REGION Network 42: MB3 Code 4082 - REGOLAZ. BORDATRICE - PASSAGGIO 02 - LATO-OP
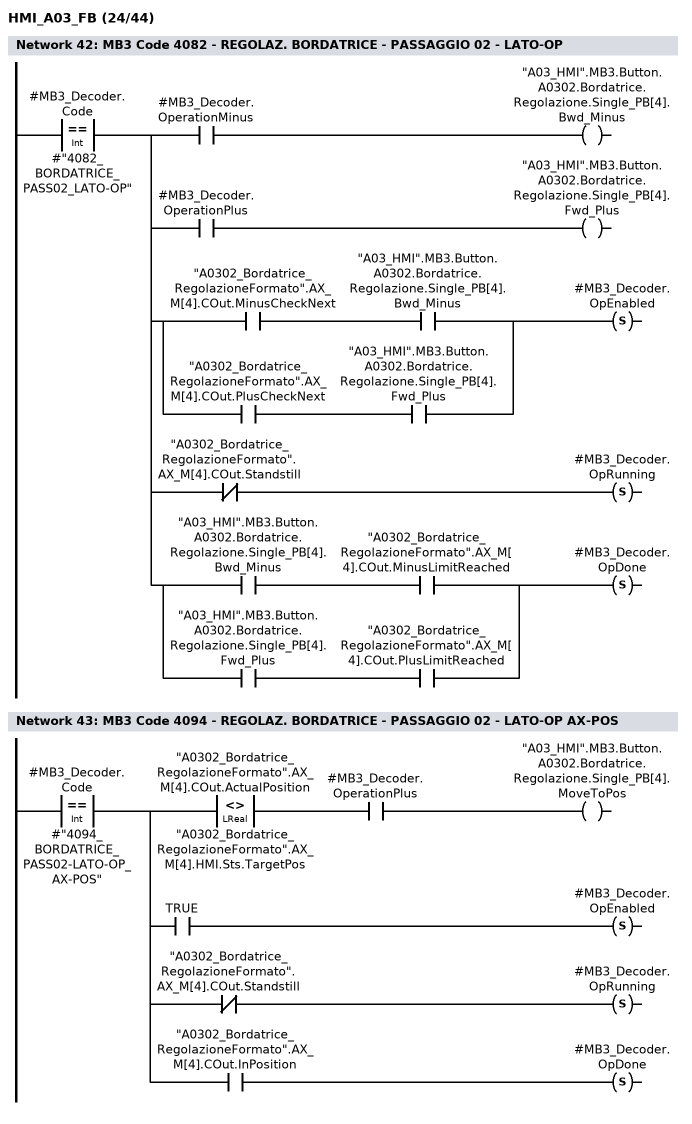
   RUNG wire#powerrail
      { S7_Templates := "SrcType := Int" } EQ_Contact(in1 := #MB3_Decoder.Code, in2 := #"4082_BORDATRICE_PASS02_LATO-OP")
      wire#w1
      Contact( #MB3_Decoder.OperationMinus )
      Coil( "A03_HMI".MB3.Button.A0302.Bordatrice.Regolazione.Single_PB[4].Bwd_Minus )
   END_RUNG
   RUNG wire#w1
      Contact( #MB3_Decoder.OperationPlus )
      Coil( "A03_HMI".MB3.Button.A0302.Bordatrice.Regolazione.Single_PB[4].Fwd_Plus )
   END_RUNG
   RUNG wire#w1
      Contact( "A0302_Bordatrice_RegolazioneFormato".AX_M[4].COut.MinusCheckNext )
      Contact( "A03_HMI".MB3.Button.A0302.Bordatrice.Regolazione.Single_PB[4].Bwd_Minus )
      wire#w2
      S_Coil( #MB3_Decoder.OpEnabled )
   END_RUNG
   RUNG wire#w1
      Contact( "A0302_Bordatrice_RegolazioneFormato".AX_M[4].COut.PlusCheckNext )
      Contact( "A03_HMI".MB3.Button.A0302.Bordatrice.Regolazione.Single_PB[4].Fwd_Plus )
   END_RUNG wire#w2
   RUNG wire#w1
      I_Contact( "A0302_Bordatrice_RegolazioneFormato".AX_M[4].COut.Standstill )
      S_Coil( #MB3_Decoder.OpRunning )
   END_RUNG
   RUNG wire#w1
      Contact( "A03_HMI".MB3.Button.A0302.Bordatrice.Regolazione.Single_PB[4].Bwd_Minus )
      Contact( "A0302_Bordatrice_RegolazioneFormato".AX_M[4].COut.MinusLimitReached )
      wire#w3
      S_Coil( #MB3_Decoder.OpDone )
   END_RUNG
   RUNG wire#w1
      Contact( "A03_HMI".MB3.Button.A0302.Bordatrice.Regolazione.Single_PB[4].Fwd_Plus )
      Contact( "A0302_Bordatrice_RegolazioneFormato".AX_M[4].COut.PlusLimitReached )
   END_RUNG wire#w3
   // the same network as SCL:
   #_w1 := #MB3_Decoder.Code = #"4082_BORDATRICE_PASS02_LATO-OP";
   "A03_HMI".MB3.Button.A0302.Bordatrice.Regolazione.Single_PB[4].Bwd_Minus := #_w1 AND #MB3_Decoder.OperationMinus;
   "A03_HMI".MB3.Button.A0302.Bordatrice.Regolazione.Single_PB[4].Fwd_Plus := #_w1 AND #MB3_Decoder.OperationPlus;
   IF #_w1 AND (("A0302_Bordatrice_RegolazioneFormato".AX_M[4].COut.MinusCheckNext AND "A03_HMI".MB3.Button.A0302.Bordatrice.Regolazione.Single_PB[4].Bwd_Minus) OR ("A0302_Bordatrice_RegolazioneFormato".AX_M[4].COut.PlusCheckNext AND "A03_HMI".MB3.Button.A0302.Bordatrice.Regolazione.Single_PB[4].Fwd_Plus)) THEN
       #MB3_Decoder.OpEnabled := TRUE;
   END_IF;
   IF #_w1 AND NOT "A0302_Bordatrice_RegolazioneFormato".AX_M[4].COut.Standstill THEN
       #MB3_Decoder.OpRunning := TRUE;
   END_IF;
   IF #_w1 AND (("A03_HMI".MB3.Button.A0302.Bordatrice.Regolazione.Single_PB[4].Bwd_Minus AND "A0302_Bordatrice_RegolazioneFormato".AX_M[4].COut.MinusLimitReached) OR ("A03_HMI".MB3.Button.A0302.Bordatrice.Regolazione.Single_PB[4].Fwd_Plus AND "A0302_Bordatrice_RegolazioneFormato".AX_M[4].COut.PlusLimitReached)) THEN
       #MB3_Decoder.OpDone := TRUE;
   END_IF;
END_REGION

REGION Network 43: MB3 Code 4094 - REGOLAZ. BORDATRICE - PASSAGGIO 02 - LATO-OP AX-POS
   RUNG wire#powerrail
      { S7_Templates := "SrcType := Int" } EQ_Contact(in1 := #MB3_Decoder.Code, in2 := #"4094_BORDATRICE_PASS02-LATO-OP_AX-POS")
      wire#w1
      { S7_Templates := "SrcType := LReal" } NE_Contact(in1 := "A0302_Bordatrice_RegolazioneFormato".AX_M[4].COut.ActualPosition, in2 := "A0302_Bordatrice_RegolazioneFormato".AX_M[4].HMI.Sts.TargetPos)
      Contact( #MB3_Decoder.OperationPlus )
      Coil( "A03_HMI".MB3.Button.A0302.Bordatrice.Regolazione.Single_PB[4].MoveToPos )
   END_RUNG
   RUNG wire#w1
      Contact( TRUE )
      S_Coil( #MB3_Decoder.OpEnabled )
   END_RUNG
   RUNG wire#w1
      I_Contact( "A0302_Bordatrice_RegolazioneFormato".AX_M[4].COut.Standstill )
      S_Coil( #MB3_Decoder.OpRunning )
   END_RUNG
   RUNG wire#w1
      Contact( "A0302_Bordatrice_RegolazioneFormato".AX_M[4].COut.InPosition )
      S_Coil( #MB3_Decoder.OpDone )
   END_RUNG
   // the same network as SCL:
   #_w1 := #MB3_Decoder.Code = #"4094_BORDATRICE_PASS02-LATO-OP_AX-POS";
   "A03_HMI".MB3.Button.A0302.Bordatrice.Regolazione.Single_PB[4].MoveToPos := #_w1 AND ("A0302_Bordatrice_RegolazioneFormato".AX_M[4].COut.ActualPosition <> "A0302_Bordatrice_RegolazioneFormato".AX_M[4].HMI.Sts.TargetPos) AND #MB3_Decoder.OperationPlus;
   IF #_w1 AND TRUE THEN #MB3_Decoder.OpEnabled := TRUE; END_IF;
   IF #_w1 AND NOT "A0302_Bordatrice_RegolazioneFormato".AX_M[4].COut.Standstill THEN
       #MB3_Decoder.OpRunning := TRUE;
   END_IF;
   IF #_w1 AND "A0302_Bordatrice_RegolazioneFormato".AX_M[4].COut.InPosition THEN
       #MB3_Decoder.OpDone := TRUE;
   END_IF;
END_REGION

REGION Network 44: MB3 Code 4083 - REGOLAZ. BORDATRICE - PASSAGGIO 02 - LATO-MOT
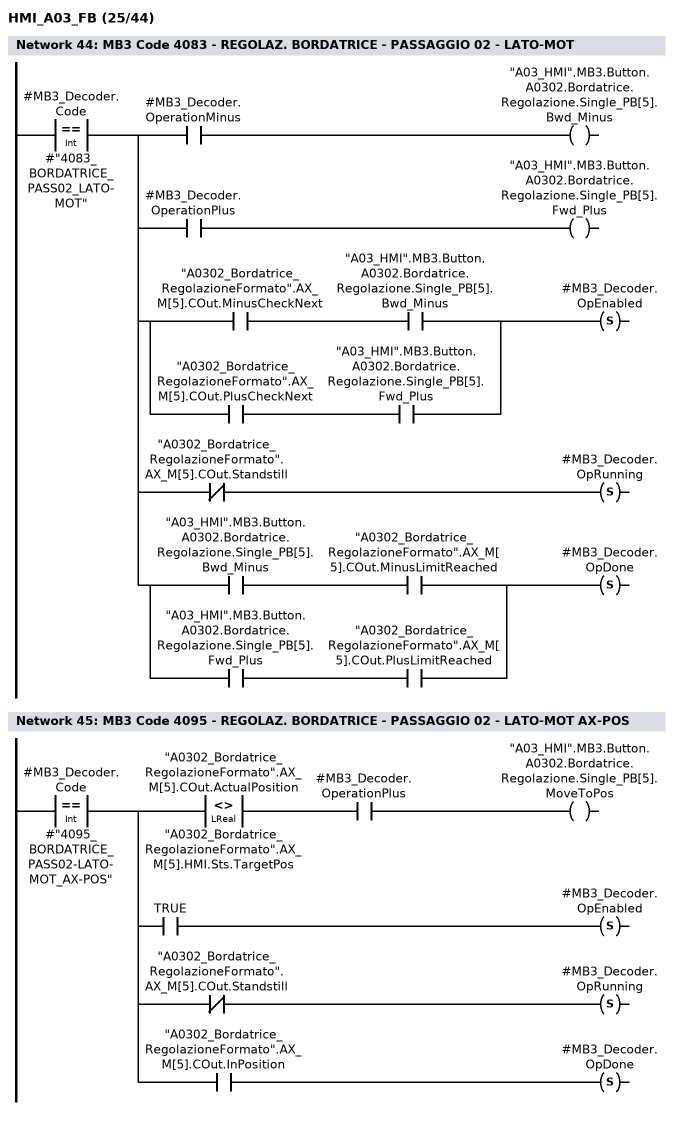
   RUNG wire#powerrail
      { S7_Templates := "SrcType := Int" } EQ_Contact(in1 := #MB3_Decoder.Code, in2 := #"4083_BORDATRICE_PASS02_LATO-MOT")
      wire#w1
      Contact( #MB3_Decoder.OperationMinus )
      Coil( "A03_HMI".MB3.Button.A0302.Bordatrice.Regolazione.Single_PB[5].Bwd_Minus )
   END_RUNG
   RUNG wire#w1
      Contact( #MB3_Decoder.OperationPlus )
      Coil( "A03_HMI".MB3.Button.A0302.Bordatrice.Regolazione.Single_PB[5].Fwd_Plus )
   END_RUNG
   RUNG wire#w1
      Contact( "A0302_Bordatrice_RegolazioneFormato".AX_M[5].COut.MinusCheckNext )
      Contact( "A03_HMI".MB3.Button.A0302.Bordatrice.Regolazione.Single_PB[5].Bwd_Minus )
      wire#w2
      S_Coil( #MB3_Decoder.OpEnabled )
   END_RUNG
   RUNG wire#w1
      Contact( "A0302_Bordatrice_RegolazioneFormato".AX_M[5].COut.PlusCheckNext )
      Contact( "A03_HMI".MB3.Button.A0302.Bordatrice.Regolazione.Single_PB[5].Fwd_Plus )
   END_RUNG wire#w2
   RUNG wire#w1
      I_Contact( "A0302_Bordatrice_RegolazioneFormato".AX_M[5].COut.Standstill )
      S_Coil( #MB3_Decoder.OpRunning )
   END_RUNG
   RUNG wire#w1
      Contact( "A03_HMI".MB3.Button.A0302.Bordatrice.Regolazione.Single_PB[5].Bwd_Minus )
      Contact( "A0302_Bordatrice_RegolazioneFormato".AX_M[5].COut.MinusLimitReached )
      wire#w3
      S_Coil( #MB3_Decoder.OpDone )
   END_RUNG
   RUNG wire#w1
      Contact( "A03_HMI".MB3.Button.A0302.Bordatrice.Regolazione.Single_PB[5].Fwd_Plus )
      Contact( "A0302_Bordatrice_RegolazioneFormato".AX_M[5].COut.PlusLimitReached )
   END_RUNG wire#w3
   // the same network as SCL:
   #_w1 := #MB3_Decoder.Code = #"4083_BORDATRICE_PASS02_LATO-MOT";
   "A03_HMI".MB3.Button.A0302.Bordatrice.Regolazione.Single_PB[5].Bwd_Minus := #_w1 AND #MB3_Decoder.OperationMinus;
   "A03_HMI".MB3.Button.A0302.Bordatrice.Regolazione.Single_PB[5].Fwd_Plus := #_w1 AND #MB3_Decoder.OperationPlus;
   IF #_w1 AND (("A0302_Bordatrice_RegolazioneFormato".AX_M[5].COut.MinusCheckNext AND "A03_HMI".MB3.Button.A0302.Bordatrice.Regolazione.Single_PB[5].Bwd_Minus) OR ("A0302_Bordatrice_RegolazioneFormato".AX_M[5].COut.PlusCheckNext AND "A03_HMI".MB3.Button.A0302.Bordatrice.Regolazione.Single_PB[5].Fwd_Plus)) THEN
       #MB3_Decoder.OpEnabled := TRUE;
   END_IF;
   IF #_w1 AND NOT "A0302_Bordatrice_RegolazioneFormato".AX_M[5].COut.Standstill THEN
       #MB3_Decoder.OpRunning := TRUE;
   END_IF;
   IF #_w1 AND (("A03_HMI".MB3.Button.A0302.Bordatrice.Regolazione.Single_PB[5].Bwd_Minus AND "A0302_Bordatrice_RegolazioneFormato".AX_M[5].COut.MinusLimitReached) OR ("A03_HMI".MB3.Button.A0302.Bordatrice.Regolazione.Single_PB[5].Fwd_Plus AND "A0302_Bordatrice_RegolazioneFormato".AX_M[5].COut.PlusLimitReached)) THEN
       #MB3_Decoder.OpDone := TRUE;
   END_IF;
END_REGION

REGION Network 45: MB3 Code 4095 - REGOLAZ. BORDATRICE - PASSAGGIO 02 - LATO-MOT AX-POS
   RUNG wire#powerrail
      { S7_Templates := "SrcType := Int" } EQ_Contact(in1 := #MB3_Decoder.Code, in2 := #"4095_BORDATRICE_PASS02-LATO-MOT_AX-POS")
      wire#w1
      { S7_Templates := "SrcType := LReal" } NE_Contact(in1 := "A0302_Bordatrice_RegolazioneFormato".AX_M[5].COut.ActualPosition, in2 := "A0302_Bordatrice_RegolazioneFormato".AX_M[5].HMI.Sts.TargetPos)
      Contact( #MB3_Decoder.OperationPlus )
      Coil( "A03_HMI".MB3.Button.A0302.Bordatrice.Regolazione.Single_PB[5].MoveToPos )
   END_RUNG
   RUNG wire#w1
      Contact( TRUE )
      S_Coil( #MB3_Decoder.OpEnabled )
   END_RUNG
   RUNG wire#w1
      I_Contact( "A0302_Bordatrice_RegolazioneFormato".AX_M[5].COut.Standstill )
      S_Coil( #MB3_Decoder.OpRunning )
   END_RUNG
   RUNG wire#w1
      Contact( "A0302_Bordatrice_RegolazioneFormato".AX_M[5].COut.InPosition )
      S_Coil( #MB3_Decoder.OpDone )
   END_RUNG
   // the same network as SCL:
   #_w1 := #MB3_Decoder.Code = #"4095_BORDATRICE_PASS02-LATO-MOT_AX-POS";
   "A03_HMI".MB3.Button.A0302.Bordatrice.Regolazione.Single_PB[5].MoveToPos := #_w1 AND ("A0302_Bordatrice_RegolazioneFormato".AX_M[5].COut.ActualPosition <> "A0302_Bordatrice_RegolazioneFormato".AX_M[5].HMI.Sts.TargetPos) AND #MB3_Decoder.OperationPlus;
   IF #_w1 AND TRUE THEN #MB3_Decoder.OpEnabled := TRUE; END_IF;
   IF #_w1 AND NOT "A0302_Bordatrice_RegolazioneFormato".AX_M[5].COut.Standstill THEN
       #MB3_Decoder.OpRunning := TRUE;
   END_IF;
   IF #_w1 AND "A0302_Bordatrice_RegolazioneFormato".AX_M[5].COut.InPosition THEN
       #MB3_Decoder.OpDone := TRUE;
   END_IF;
END_REGION

REGION Network 46: MB3 Code 4036 - REGOLAZ. BORDATRICE - PASSAGGIO 03 - COMBO
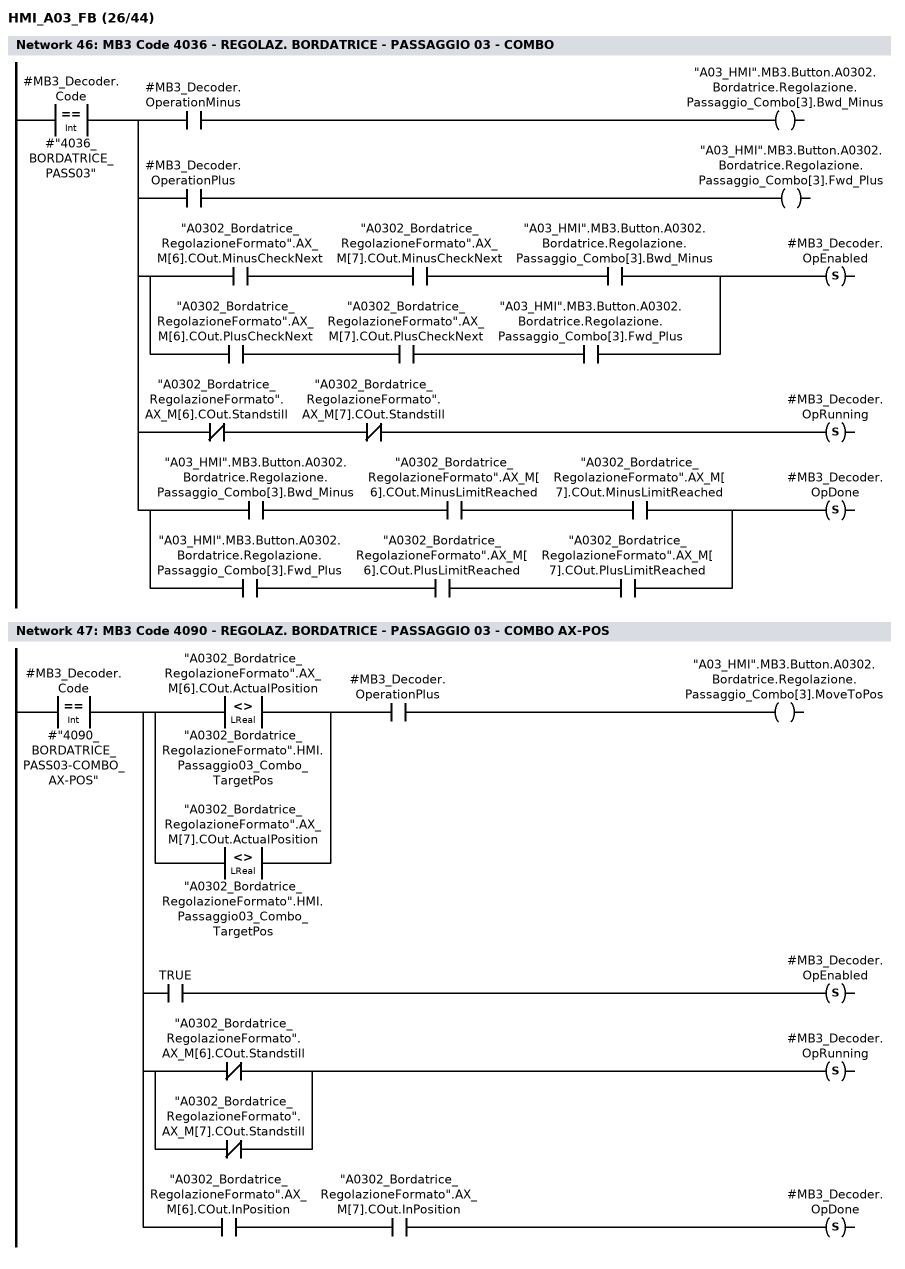
   RUNG wire#powerrail
      { S7_Templates := "SrcType := Int" } EQ_Contact(in1 := #MB3_Decoder.Code, in2 := #"4036_BORDATRICE_PASS03")
      wire#w1
      Contact( #MB3_Decoder.OperationMinus )
      Coil( "A03_HMI".MB3.Button.A0302.Bordatrice.Regolazione.Passaggio_Combo[3].Bwd_Minus )
   END_RUNG
   RUNG wire#w1
      Contact( #MB3_Decoder.OperationPlus )
      Coil( "A03_HMI".MB3.Button.A0302.Bordatrice.Regolazione.Passaggio_Combo[3].Fwd_Plus )
   END_RUNG
   RUNG wire#w1
      Contact( "A0302_Bordatrice_RegolazioneFormato".AX_M[6].COut.MinusCheckNext )
      Contact( "A0302_Bordatrice_RegolazioneFormato".AX_M[7].COut.MinusCheckNext )
      Contact( "A03_HMI".MB3.Button.A0302.Bordatrice.Regolazione.Passaggio_Combo[3].Bwd_Minus )
      wire#w2
      S_Coil( #MB3_Decoder.OpEnabled )
   END_RUNG
   RUNG wire#w1
      Contact( "A0302_Bordatrice_RegolazioneFormato".AX_M[6].COut.PlusCheckNext )
      Contact( "A0302_Bordatrice_RegolazioneFormato".AX_M[7].COut.PlusCheckNext )
      Contact( "A03_HMI".MB3.Button.A0302.Bordatrice.Regolazione.Passaggio_Combo[3].Fwd_Plus )
   END_RUNG wire#w2
   RUNG wire#w1
      I_Contact( "A0302_Bordatrice_RegolazioneFormato".AX_M[6].COut.Standstill )
      I_Contact( "A0302_Bordatrice_RegolazioneFormato".AX_M[7].COut.Standstill )
      S_Coil( #MB3_Decoder.OpRunning )
   END_RUNG
   RUNG wire#w1
      Contact( "A03_HMI".MB3.Button.A0302.Bordatrice.Regolazione.Passaggio_Combo[3].Bwd_Minus )
      Contact( "A0302_Bordatrice_RegolazioneFormato".AX_M[6].COut.MinusLimitReached )
      Contact( "A0302_Bordatrice_RegolazioneFormato".AX_M[7].COut.MinusLimitReached )
      wire#w3
      S_Coil( #MB3_Decoder.OpDone )
   END_RUNG
   RUNG wire#w1
      Contact( "A03_HMI".MB3.Button.A0302.Bordatrice.Regolazione.Passaggio_Combo[3].Fwd_Plus )
      Contact( "A0302_Bordatrice_RegolazioneFormato".AX_M[6].COut.PlusLimitReached )
      Contact( "A0302_Bordatrice_RegolazioneFormato".AX_M[7].COut.PlusLimitReached )
   END_RUNG wire#w3
   // the same network as SCL:
   #_w1 := #MB3_Decoder.Code = #"4036_BORDATRICE_PASS03";
   "A03_HMI".MB3.Button.A0302.Bordatrice.Regolazione.Passaggio_Combo[3].Bwd_Minus := #_w1 AND #MB3_Decoder.OperationMinus;
   "A03_HMI".MB3.Button.A0302.Bordatrice.Regolazione.Passaggio_Combo[3].Fwd_Plus := #_w1 AND #MB3_Decoder.OperationPlus;
   IF #_w1 AND (("A0302_Bordatrice_RegolazioneFormato".AX_M[6].COut.MinusCheckNext AND "A0302_Bordatrice_RegolazioneFormato".AX_M[7].COut.MinusCheckNext AND "A03_HMI".MB3.Button.A0302.Bordatrice.Regolazione.Passaggio_Combo[3].Bwd_Minus) OR ("A0302_Bordatrice_RegolazioneFormato".AX_M[6].COut.PlusCheckNext AND "A0302_Bordatrice_RegolazioneFormato".AX_M[7].COut.PlusCheckNext AND "A03_HMI".MB3.Button.A0302.Bordatrice.Regolazione.Passaggio_Combo[3].Fwd_Plus)) THEN
       #MB3_Decoder.OpEnabled := TRUE;
   END_IF;
   IF #_w1 AND NOT "A0302_Bordatrice_RegolazioneFormato".AX_M[6].COut.Standstill AND NOT "A0302_Bordatrice_RegolazioneFormato".AX_M[7].COut.Standstill THEN
       #MB3_Decoder.OpRunning := TRUE;
   END_IF;
   IF #_w1 AND (("A03_HMI".MB3.Button.A0302.Bordatrice.Regolazione.Passaggio_Combo[3].Bwd_Minus AND "A0302_Bordatrice_RegolazioneFormato".AX_M[6].COut.MinusLimitReached AND "A0302_Bordatrice_RegolazioneFormato".AX_M[7].COut.MinusLimitReached) OR ("A03_HMI".MB3.Button.A0302.Bordatrice.Regolazione.Passaggio_Combo[3].Fwd_Plus AND "A0302_Bordatrice_RegolazioneFormato".AX_M[6].COut.PlusLimitReached AND "A0302_Bordatrice_RegolazioneFormato".AX_M[7].COut.PlusLimitReached)) THEN
       #MB3_Decoder.OpDone := TRUE;
   END_IF;
END_REGION

REGION Network 47: MB3 Code 4090 - REGOLAZ. BORDATRICE - PASSAGGIO 03 - COMBO AX-POS
   RUNG wire#powerrail
      { S7_Templates := "SrcType := Int" } EQ_Contact(in1 := #MB3_Decoder.Code, in2 := #"4090_BORDATRICE_PASS03-COMBO_AX-POS")
      wire#w1
      { S7_Templates := "SrcType := LReal" } NE_Contact(in1 := "A0302_Bordatrice_RegolazioneFormato".AX_M[6].COut.ActualPosition, in2 := "A0302_Bordatrice_RegolazioneFormato".HMI.Passaggio03_Combo_TargetPos)
      wire#w2
      Contact( #MB3_Decoder.OperationPlus )
      Coil( "A03_HMI".MB3.Button.A0302.Bordatrice.Regolazione.Passaggio_Combo[3].MoveToPos )
   END_RUNG
   RUNG wire#w1
      { S7_Templates := "SrcType := LReal" } NE_Contact(in1 := "A0302_Bordatrice_RegolazioneFormato".AX_M[7].COut.ActualPosition, in2 := "A0302_Bordatrice_RegolazioneFormato".HMI.Passaggio03_Combo_TargetPos)
   END_RUNG wire#w2
   RUNG wire#w1
      Contact( TRUE )
      S_Coil( #MB3_Decoder.OpEnabled )
   END_RUNG
   RUNG wire#w1
      I_Contact( "A0302_Bordatrice_RegolazioneFormato".AX_M[6].COut.Standstill )
      wire#w3
      S_Coil( #MB3_Decoder.OpRunning )
   END_RUNG
   RUNG wire#w1
      I_Contact( "A0302_Bordatrice_RegolazioneFormato".AX_M[7].COut.Standstill )
   END_RUNG wire#w3
   RUNG wire#w1
      Contact( "A0302_Bordatrice_RegolazioneFormato".AX_M[6].COut.InPosition )
      Contact( "A0302_Bordatrice_RegolazioneFormato".AX_M[7].COut.InPosition )
      S_Coil( #MB3_Decoder.OpDone )
   END_RUNG
   // the same network as SCL:
   #_w1 := #MB3_Decoder.Code = #"4090_BORDATRICE_PASS03-COMBO_AX-POS";
   "A03_HMI".MB3.Button.A0302.Bordatrice.Regolazione.Passaggio_Combo[3].MoveToPos := #_w1 AND (("A0302_Bordatrice_RegolazioneFormato".AX_M[6].COut.ActualPosition <> "A0302_Bordatrice_RegolazioneFormato".HMI.Passaggio03_Combo_TargetPos) OR ("A0302_Bordatrice_RegolazioneFormato".AX_M[7].COut.ActualPosition <> "A0302_Bordatrice_RegolazioneFormato".HMI.Passaggio03_Combo_TargetPos)) AND #MB3_Decoder.OperationPlus;
   IF #_w1 AND TRUE THEN #MB3_Decoder.OpEnabled := TRUE; END_IF;
   IF #_w1 AND (NOT "A0302_Bordatrice_RegolazioneFormato".AX_M[6].COut.Standstill OR NOT "A0302_Bordatrice_RegolazioneFormato".AX_M[7].COut.Standstill) THEN
       #MB3_Decoder.OpRunning := TRUE;
   END_IF;
   IF #_w1 AND "A0302_Bordatrice_RegolazioneFormato".AX_M[6].COut.InPosition AND "A0302_Bordatrice_RegolazioneFormato".AX_M[7].COut.InPosition THEN
       #MB3_Decoder.OpDone := TRUE;
   END_IF;
END_REGION

REGION Network 48: MB3 Code 4084 - REGOLAZ. BORDATRICE - PASSAGGIO 03 - LATO-OP
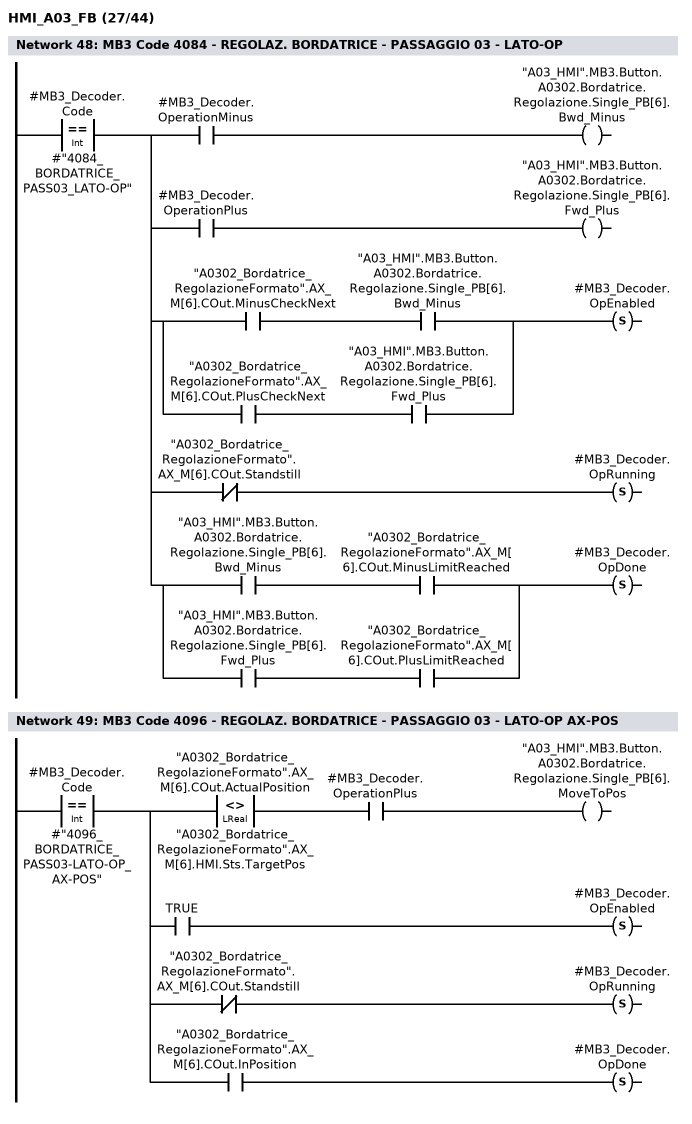
   RUNG wire#powerrail
      { S7_Templates := "SrcType := Int" } EQ_Contact(in1 := #MB3_Decoder.Code, in2 := #"4084_BORDATRICE_PASS03_LATO-OP")
      wire#w1
      Contact( #MB3_Decoder.OperationMinus )
      Coil( "A03_HMI".MB3.Button.A0302.Bordatrice.Regolazione.Single_PB[6].Bwd_Minus )
   END_RUNG
   RUNG wire#w1
      Contact( #MB3_Decoder.OperationPlus )
      Coil( "A03_HMI".MB3.Button.A0302.Bordatrice.Regolazione.Single_PB[6].Fwd_Plus )
   END_RUNG
   RUNG wire#w1
      Contact( "A0302_Bordatrice_RegolazioneFormato".AX_M[6].COut.MinusCheckNext )
      Contact( "A03_HMI".MB3.Button.A0302.Bordatrice.Regolazione.Single_PB[6].Bwd_Minus )
      wire#w2
      S_Coil( #MB3_Decoder.OpEnabled )
   END_RUNG
   RUNG wire#w1
      Contact( "A0302_Bordatrice_RegolazioneFormato".AX_M[6].COut.PlusCheckNext )
      Contact( "A03_HMI".MB3.Button.A0302.Bordatrice.Regolazione.Single_PB[6].Fwd_Plus )
   END_RUNG wire#w2
   RUNG wire#w1
      I_Contact( "A0302_Bordatrice_RegolazioneFormato".AX_M[6].COut.Standstill )
      S_Coil( #MB3_Decoder.OpRunning )
   END_RUNG
   RUNG wire#w1
      Contact( "A03_HMI".MB3.Button.A0302.Bordatrice.Regolazione.Single_PB[6].Bwd_Minus )
      Contact( "A0302_Bordatrice_RegolazioneFormato".AX_M[6].COut.MinusLimitReached )
      wire#w3
      S_Coil( #MB3_Decoder.OpDone )
   END_RUNG
   RUNG wire#w1
      Contact( "A03_HMI".MB3.Button.A0302.Bordatrice.Regolazione.Single_PB[6].Fwd_Plus )
      Contact( "A0302_Bordatrice_RegolazioneFormato".AX_M[6].COut.PlusLimitReached )
   END_RUNG wire#w3
   // the same network as SCL:
   #_w1 := #MB3_Decoder.Code = #"4084_BORDATRICE_PASS03_LATO-OP";
   "A03_HMI".MB3.Button.A0302.Bordatrice.Regolazione.Single_PB[6].Bwd_Minus := #_w1 AND #MB3_Decoder.OperationMinus;
   "A03_HMI".MB3.Button.A0302.Bordatrice.Regolazione.Single_PB[6].Fwd_Plus := #_w1 AND #MB3_Decoder.OperationPlus;
   IF #_w1 AND (("A0302_Bordatrice_RegolazioneFormato".AX_M[6].COut.MinusCheckNext AND "A03_HMI".MB3.Button.A0302.Bordatrice.Regolazione.Single_PB[6].Bwd_Minus) OR ("A0302_Bordatrice_RegolazioneFormato".AX_M[6].COut.PlusCheckNext AND "A03_HMI".MB3.Button.A0302.Bordatrice.Regolazione.Single_PB[6].Fwd_Plus)) THEN
       #MB3_Decoder.OpEnabled := TRUE;
   END_IF;
   IF #_w1 AND NOT "A0302_Bordatrice_RegolazioneFormato".AX_M[6].COut.Standstill THEN
       #MB3_Decoder.OpRunning := TRUE;
   END_IF;
   IF #_w1 AND (("A03_HMI".MB3.Button.A0302.Bordatrice.Regolazione.Single_PB[6].Bwd_Minus AND "A0302_Bordatrice_RegolazioneFormato".AX_M[6].COut.MinusLimitReached) OR ("A03_HMI".MB3.Button.A0302.Bordatrice.Regolazione.Single_PB[6].Fwd_Plus AND "A0302_Bordatrice_RegolazioneFormato".AX_M[6].COut.PlusLimitReached)) THEN
       #MB3_Decoder.OpDone := TRUE;
   END_IF;
END_REGION

REGION Network 49: MB3 Code 4096 - REGOLAZ. BORDATRICE - PASSAGGIO 03 - LATO-OP AX-POS
   RUNG wire#powerrail
      { S7_Templates := "SrcType := Int" } EQ_Contact(in1 := #MB3_Decoder.Code, in2 := #"4096_BORDATRICE_PASS03-LATO-OP_AX-POS")
      wire#w1
      { S7_Templates := "SrcType := LReal" } NE_Contact(in1 := "A0302_Bordatrice_RegolazioneFormato".AX_M[6].COut.ActualPosition, in2 := "A0302_Bordatrice_RegolazioneFormato".AX_M[6].HMI.Sts.TargetPos)
      Contact( #MB3_Decoder.OperationPlus )
      Coil( "A03_HMI".MB3.Button.A0302.Bordatrice.Regolazione.Single_PB[6].MoveToPos )
   END_RUNG
   RUNG wire#w1
      Contact( TRUE )
      S_Coil( #MB3_Decoder.OpEnabled )
   END_RUNG
   RUNG wire#w1
      I_Contact( "A0302_Bordatrice_RegolazioneFormato".AX_M[6].COut.Standstill )
      S_Coil( #MB3_Decoder.OpRunning )
   END_RUNG
   RUNG wire#w1
      Contact( "A0302_Bordatrice_RegolazioneFormato".AX_M[6].COut.InPosition )
      S_Coil( #MB3_Decoder.OpDone )
   END_RUNG
   // the same network as SCL:
   #_w1 := #MB3_Decoder.Code = #"4096_BORDATRICE_PASS03-LATO-OP_AX-POS";
   "A03_HMI".MB3.Button.A0302.Bordatrice.Regolazione.Single_PB[6].MoveToPos := #_w1 AND ("A0302_Bordatrice_RegolazioneFormato".AX_M[6].COut.ActualPosition <> "A0302_Bordatrice_RegolazioneFormato".AX_M[6].HMI.Sts.TargetPos) AND #MB3_Decoder.OperationPlus;
   IF #_w1 AND TRUE THEN #MB3_Decoder.OpEnabled := TRUE; END_IF;
   IF #_w1 AND NOT "A0302_Bordatrice_RegolazioneFormato".AX_M[6].COut.Standstill THEN
       #MB3_Decoder.OpRunning := TRUE;
   END_IF;
   IF #_w1 AND "A0302_Bordatrice_RegolazioneFormato".AX_M[6].COut.InPosition THEN
       #MB3_Decoder.OpDone := TRUE;
   END_IF;
END_REGION

REGION Network 50: MB3 Code 4085 - REGOLAZ. BORDATRICE - PASSAGGIO 03 - LATO-MOT
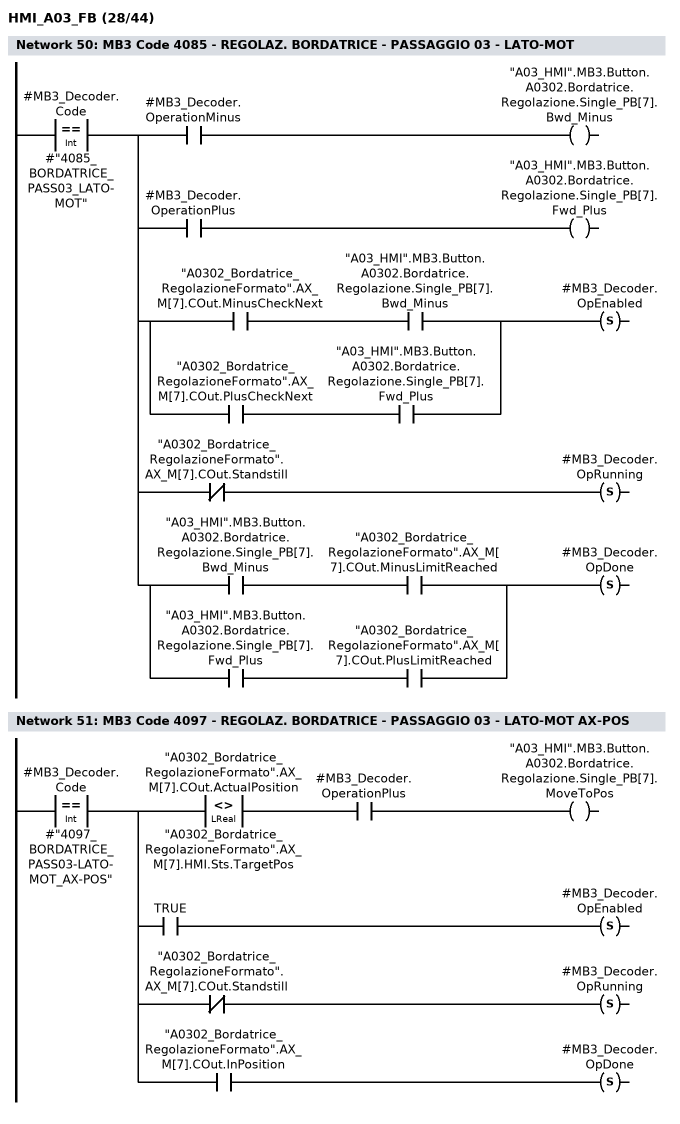
   RUNG wire#powerrail
      { S7_Templates := "SrcType := Int" } EQ_Contact(in1 := #MB3_Decoder.Code, in2 := #"4085_BORDATRICE_PASS03_LATO-MOT")
      wire#w1
      Contact( #MB3_Decoder.OperationMinus )
      Coil( "A03_HMI".MB3.Button.A0302.Bordatrice.Regolazione.Single_PB[7].Bwd_Minus )
   END_RUNG
   RUNG wire#w1
      Contact( #MB3_Decoder.OperationPlus )
      Coil( "A03_HMI".MB3.Button.A0302.Bordatrice.Regolazione.Single_PB[7].Fwd_Plus )
   END_RUNG
   RUNG wire#w1
      Contact( "A0302_Bordatrice_RegolazioneFormato".AX_M[7].COut.MinusCheckNext )
      Contact( "A03_HMI".MB3.Button.A0302.Bordatrice.Regolazione.Single_PB[7].Bwd_Minus )
      wire#w2
      S_Coil( #MB3_Decoder.OpEnabled )
   END_RUNG
   RUNG wire#w1
      Contact( "A0302_Bordatrice_RegolazioneFormato".AX_M[7].COut.PlusCheckNext )
      Contact( "A03_HMI".MB3.Button.A0302.Bordatrice.Regolazione.Single_PB[7].Fwd_Plus )
   END_RUNG wire#w2
   RUNG wire#w1
      I_Contact( "A0302_Bordatrice_RegolazioneFormato".AX_M[7].COut.Standstill )
      S_Coil( #MB3_Decoder.OpRunning )
   END_RUNG
   RUNG wire#w1
      Contact( "A03_HMI".MB3.Button.A0302.Bordatrice.Regolazione.Single_PB[7].Bwd_Minus )
      Contact( "A0302_Bordatrice_RegolazioneFormato".AX_M[7].COut.MinusLimitReached )
      wire#w3
      S_Coil( #MB3_Decoder.OpDone )
   END_RUNG
   RUNG wire#w1
      Contact( "A03_HMI".MB3.Button.A0302.Bordatrice.Regolazione.Single_PB[7].Fwd_Plus )
      Contact( "A0302_Bordatrice_RegolazioneFormato".AX_M[7].COut.PlusLimitReached )
   END_RUNG wire#w3
   // the same network as SCL:
   #_w1 := #MB3_Decoder.Code = #"4085_BORDATRICE_PASS03_LATO-MOT";
   "A03_HMI".MB3.Button.A0302.Bordatrice.Regolazione.Single_PB[7].Bwd_Minus := #_w1 AND #MB3_Decoder.OperationMinus;
   "A03_HMI".MB3.Button.A0302.Bordatrice.Regolazione.Single_PB[7].Fwd_Plus := #_w1 AND #MB3_Decoder.OperationPlus;
   IF #_w1 AND (("A0302_Bordatrice_RegolazioneFormato".AX_M[7].COut.MinusCheckNext AND "A03_HMI".MB3.Button.A0302.Bordatrice.Regolazione.Single_PB[7].Bwd_Minus) OR ("A0302_Bordatrice_RegolazioneFormato".AX_M[7].COut.PlusCheckNext AND "A03_HMI".MB3.Button.A0302.Bordatrice.Regolazione.Single_PB[7].Fwd_Plus)) THEN
       #MB3_Decoder.OpEnabled := TRUE;
   END_IF;
   IF #_w1 AND NOT "A0302_Bordatrice_RegolazioneFormato".AX_M[7].COut.Standstill THEN
       #MB3_Decoder.OpRunning := TRUE;
   END_IF;
   IF #_w1 AND (("A03_HMI".MB3.Button.A0302.Bordatrice.Regolazione.Single_PB[7].Bwd_Minus AND "A0302_Bordatrice_RegolazioneFormato".AX_M[7].COut.MinusLimitReached) OR ("A03_HMI".MB3.Button.A0302.Bordatrice.Regolazione.Single_PB[7].Fwd_Plus AND "A0302_Bordatrice_RegolazioneFormato".AX_M[7].COut.PlusLimitReached)) THEN
       #MB3_Decoder.OpDone := TRUE;
   END_IF;
END_REGION

REGION Network 51: MB3 Code 4097 - REGOLAZ. BORDATRICE - PASSAGGIO 03 - LATO-MOT AX-POS
   RUNG wire#powerrail
      { S7_Templates := "SrcType := Int" } EQ_Contact(in1 := #MB3_Decoder.Code, in2 := #"4097_BORDATRICE_PASS03-LATO-MOT_AX-POS")
      wire#w1
      { S7_Templates := "SrcType := LReal" } NE_Contact(in1 := "A0302_Bordatrice_RegolazioneFormato".AX_M[7].COut.ActualPosition, in2 := "A0302_Bordatrice_RegolazioneFormato".AX_M[7].HMI.Sts.TargetPos)
      Contact( #MB3_Decoder.OperationPlus )
      Coil( "A03_HMI".MB3.Button.A0302.Bordatrice.Regolazione.Single_PB[7].MoveToPos )
   END_RUNG
   RUNG wire#w1
      Contact( TRUE )
      S_Coil( #MB3_Decoder.OpEnabled )
   END_RUNG
   RUNG wire#w1
      I_Contact( "A0302_Bordatrice_RegolazioneFormato".AX_M[7].COut.Standstill )
      S_Coil( #MB3_Decoder.OpRunning )
   END_RUNG
   RUNG wire#w1
      Contact( "A0302_Bordatrice_RegolazioneFormato".AX_M[7].COut.InPosition )
      S_Coil( #MB3_Decoder.OpDone )
   END_RUNG
   // the same network as SCL:
   #_w1 := #MB3_Decoder.Code = #"4097_BORDATRICE_PASS03-LATO-MOT_AX-POS";
   "A03_HMI".MB3.Button.A0302.Bordatrice.Regolazione.Single_PB[7].MoveToPos := #_w1 AND ("A0302_Bordatrice_RegolazioneFormato".AX_M[7].COut.ActualPosition <> "A0302_Bordatrice_RegolazioneFormato".AX_M[7].HMI.Sts.TargetPos) AND #MB3_Decoder.OperationPlus;
   IF #_w1 AND TRUE THEN #MB3_Decoder.OpEnabled := TRUE; END_IF;
   IF #_w1 AND NOT "A0302_Bordatrice_RegolazioneFormato".AX_M[7].COut.Standstill THEN
       #MB3_Decoder.OpRunning := TRUE;
   END_IF;
   IF #_w1 AND "A0302_Bordatrice_RegolazioneFormato".AX_M[7].COut.InPosition THEN
       #MB3_Decoder.OpDone := TRUE;
   END_IF;
END_REGION

REGION Network 52: MB3 Code 4037 - REGOLAZ. BORDATRICE - PASSAGGIO 04 - COMBO
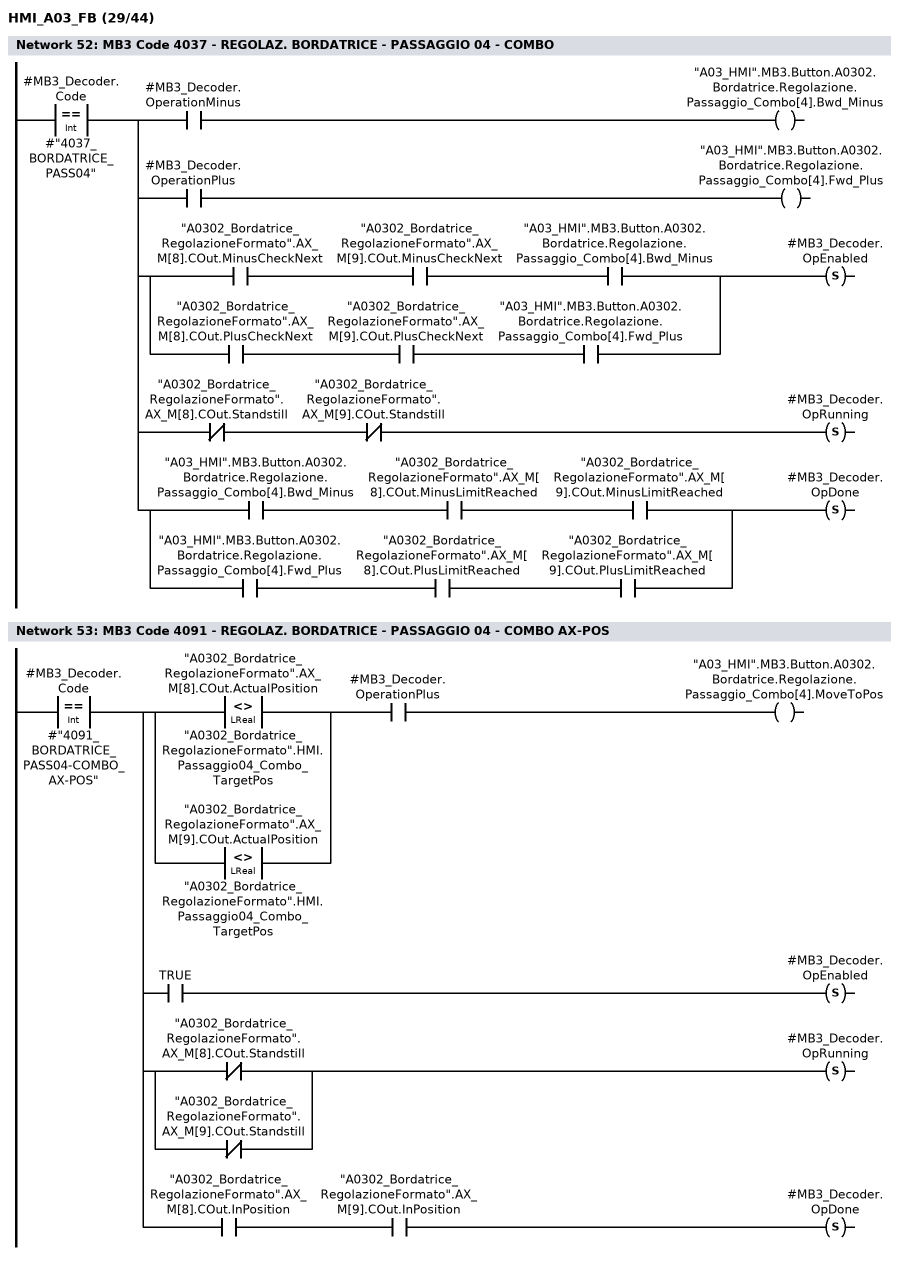
   RUNG wire#powerrail
      { S7_Templates := "SrcType := Int" } EQ_Contact(in1 := #MB3_Decoder.Code, in2 := #"4037_BORDATRICE_PASS04")
      wire#w1
      Contact( #MB3_Decoder.OperationMinus )
      Coil( "A03_HMI".MB3.Button.A0302.Bordatrice.Regolazione.Passaggio_Combo[4].Bwd_Minus )
   END_RUNG
   RUNG wire#w1
      Contact( #MB3_Decoder.OperationPlus )
      Coil( "A03_HMI".MB3.Button.A0302.Bordatrice.Regolazione.Passaggio_Combo[4].Fwd_Plus )
   END_RUNG
   RUNG wire#w1
      Contact( "A0302_Bordatrice_RegolazioneFormato".AX_M[8].COut.MinusCheckNext )
      Contact( "A0302_Bordatrice_RegolazioneFormato".AX_M[9].COut.MinusCheckNext )
      Contact( "A03_HMI".MB3.Button.A0302.Bordatrice.Regolazione.Passaggio_Combo[4].Bwd_Minus )
      wire#w2
      S_Coil( #MB3_Decoder.OpEnabled )
   END_RUNG
   RUNG wire#w1
      Contact( "A0302_Bordatrice_RegolazioneFormato".AX_M[8].COut.PlusCheckNext )
      Contact( "A0302_Bordatrice_RegolazioneFormato".AX_M[9].COut.PlusCheckNext )
      Contact( "A03_HMI".MB3.Button.A0302.Bordatrice.Regolazione.Passaggio_Combo[4].Fwd_Plus )
   END_RUNG wire#w2
   RUNG wire#w1
      I_Contact( "A0302_Bordatrice_RegolazioneFormato".AX_M[8].COut.Standstill )
      I_Contact( "A0302_Bordatrice_RegolazioneFormato".AX_M[9].COut.Standstill )
      S_Coil( #MB3_Decoder.OpRunning )
   END_RUNG
   RUNG wire#w1
      Contact( "A03_HMI".MB3.Button.A0302.Bordatrice.Regolazione.Passaggio_Combo[4].Bwd_Minus )
      Contact( "A0302_Bordatrice_RegolazioneFormato".AX_M[8].COut.MinusLimitReached )
      Contact( "A0302_Bordatrice_RegolazioneFormato".AX_M[9].COut.MinusLimitReached )
      wire#w3
      S_Coil( #MB3_Decoder.OpDone )
   END_RUNG
   RUNG wire#w1
      Contact( "A03_HMI".MB3.Button.A0302.Bordatrice.Regolazione.Passaggio_Combo[4].Fwd_Plus )
      Contact( "A0302_Bordatrice_RegolazioneFormato".AX_M[8].COut.PlusLimitReached )
      Contact( "A0302_Bordatrice_RegolazioneFormato".AX_M[9].COut.PlusLimitReached )
   END_RUNG wire#w3
   // the same network as SCL:
   #_w1 := #MB3_Decoder.Code = #"4037_BORDATRICE_PASS04";
   "A03_HMI".MB3.Button.A0302.Bordatrice.Regolazione.Passaggio_Combo[4].Bwd_Minus := #_w1 AND #MB3_Decoder.OperationMinus;
   "A03_HMI".MB3.Button.A0302.Bordatrice.Regolazione.Passaggio_Combo[4].Fwd_Plus := #_w1 AND #MB3_Decoder.OperationPlus;
   IF #_w1 AND (("A0302_Bordatrice_RegolazioneFormato".AX_M[8].COut.MinusCheckNext AND "A0302_Bordatrice_RegolazioneFormato".AX_M[9].COut.MinusCheckNext AND "A03_HMI".MB3.Button.A0302.Bordatrice.Regolazione.Passaggio_Combo[4].Bwd_Minus) OR ("A0302_Bordatrice_RegolazioneFormato".AX_M[8].COut.PlusCheckNext AND "A0302_Bordatrice_RegolazioneFormato".AX_M[9].COut.PlusCheckNext AND "A03_HMI".MB3.Button.A0302.Bordatrice.Regolazione.Passaggio_Combo[4].Fwd_Plus)) THEN
       #MB3_Decoder.OpEnabled := TRUE;
   END_IF;
   IF #_w1 AND NOT "A0302_Bordatrice_RegolazioneFormato".AX_M[8].COut.Standstill AND NOT "A0302_Bordatrice_RegolazioneFormato".AX_M[9].COut.Standstill THEN
       #MB3_Decoder.OpRunning := TRUE;
   END_IF;
   IF #_w1 AND (("A03_HMI".MB3.Button.A0302.Bordatrice.Regolazione.Passaggio_Combo[4].Bwd_Minus AND "A0302_Bordatrice_RegolazioneFormato".AX_M[8].COut.MinusLimitReached AND "A0302_Bordatrice_RegolazioneFormato".AX_M[9].COut.MinusLimitReached) OR ("A03_HMI".MB3.Button.A0302.Bordatrice.Regolazione.Passaggio_Combo[4].Fwd_Plus AND "A0302_Bordatrice_RegolazioneFormato".AX_M[8].COut.PlusLimitReached AND "A0302_Bordatrice_RegolazioneFormato".AX_M[9].COut.PlusLimitReached)) THEN
       #MB3_Decoder.OpDone := TRUE;
   END_IF;
END_REGION

REGION Network 53: MB3 Code 4091 - REGOLAZ. BORDATRICE - PASSAGGIO 04 - COMBO AX-POS
   RUNG wire#powerrail
      { S7_Templates := "SrcType := Int" } EQ_Contact(in1 := #MB3_Decoder.Code, in2 := #"4091_BORDATRICE_PASS04-COMBO_AX-POS")
      wire#w1
      { S7_Templates := "SrcType := LReal" } NE_Contact(in1 := "A0302_Bordatrice_RegolazioneFormato".AX_M[8].COut.ActualPosition, in2 := "A0302_Bordatrice_RegolazioneFormato".HMI.Passaggio04_Combo_TargetPos)
      wire#w2
      Contact( #MB3_Decoder.OperationPlus )
      Coil( "A03_HMI".MB3.Button.A0302.Bordatrice.Regolazione.Passaggio_Combo[4].MoveToPos )
   END_RUNG
   RUNG wire#w1
      { S7_Templates := "SrcType := LReal" } NE_Contact(in1 := "A0302_Bordatrice_RegolazioneFormato".AX_M[9].COut.ActualPosition, in2 := "A0302_Bordatrice_RegolazioneFormato".HMI.Passaggio04_Combo_TargetPos)
   END_RUNG wire#w2
   RUNG wire#w1
      Contact( TRUE )
      S_Coil( #MB3_Decoder.OpEnabled )
   END_RUNG
   RUNG wire#w1
      I_Contact( "A0302_Bordatrice_RegolazioneFormato".AX_M[8].COut.Standstill )
      wire#w3
      S_Coil( #MB3_Decoder.OpRunning )
   END_RUNG
   RUNG wire#w1
      I_Contact( "A0302_Bordatrice_RegolazioneFormato".AX_M[9].COut.Standstill )
   END_RUNG wire#w3
   RUNG wire#w1
      Contact( "A0302_Bordatrice_RegolazioneFormato".AX_M[8].COut.InPosition )
      Contact( "A0302_Bordatrice_RegolazioneFormato".AX_M[9].COut.InPosition )
      S_Coil( #MB3_Decoder.OpDone )
   END_RUNG
   // the same network as SCL:
   #_w1 := #MB3_Decoder.Code = #"4091_BORDATRICE_PASS04-COMBO_AX-POS";
   "A03_HMI".MB3.Button.A0302.Bordatrice.Regolazione.Passaggio_Combo[4].MoveToPos := #_w1 AND (("A0302_Bordatrice_RegolazioneFormato".AX_M[8].COut.ActualPosition <> "A0302_Bordatrice_RegolazioneFormato".HMI.Passaggio04_Combo_TargetPos) OR ("A0302_Bordatrice_RegolazioneFormato".AX_M[9].COut.ActualPosition <> "A0302_Bordatrice_RegolazioneFormato".HMI.Passaggio04_Combo_TargetPos)) AND #MB3_Decoder.OperationPlus;
   IF #_w1 AND TRUE THEN #MB3_Decoder.OpEnabled := TRUE; END_IF;
   IF #_w1 AND (NOT "A0302_Bordatrice_RegolazioneFormato".AX_M[8].COut.Standstill OR NOT "A0302_Bordatrice_RegolazioneFormato".AX_M[9].COut.Standstill) THEN
       #MB3_Decoder.OpRunning := TRUE;
   END_IF;
   IF #_w1 AND "A0302_Bordatrice_RegolazioneFormato".AX_M[8].COut.InPosition AND "A0302_Bordatrice_RegolazioneFormato".AX_M[9].COut.InPosition THEN
       #MB3_Decoder.OpDone := TRUE;
   END_IF;
END_REGION

REGION Network 54: MB3 Code 4086 - REGOLAZ. BORDATRICE - PASSAGGIO 04 - LATO-OP
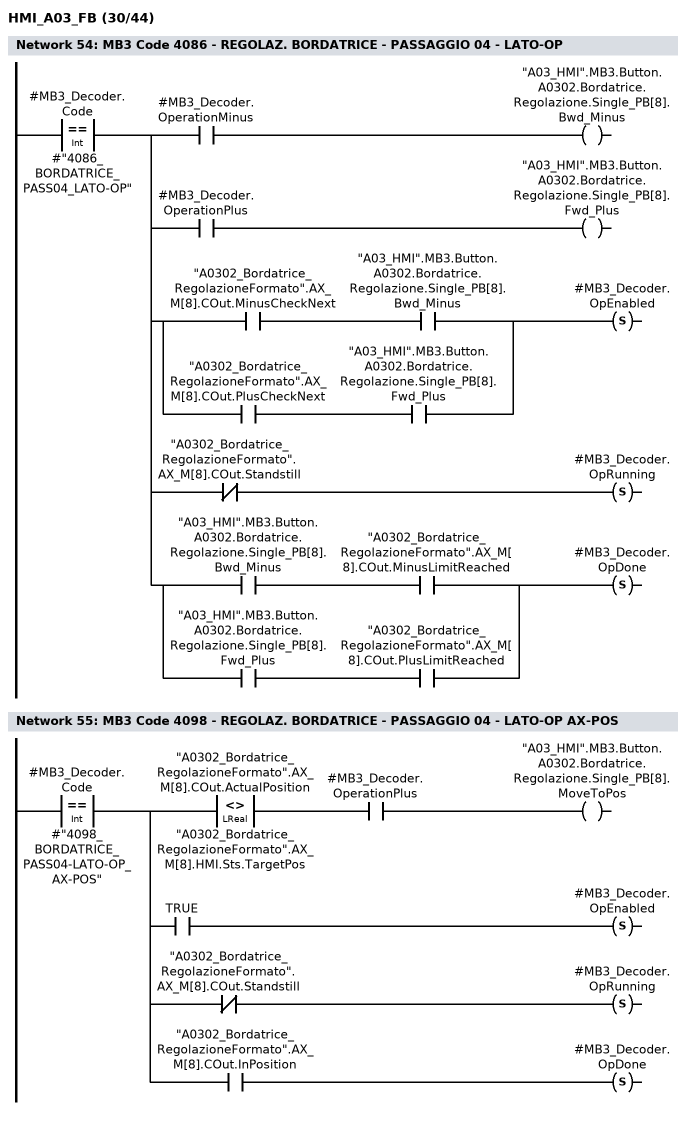
   RUNG wire#powerrail
      { S7_Templates := "SrcType := Int" } EQ_Contact(in1 := #MB3_Decoder.Code, in2 := #"4086_BORDATRICE_PASS04_LATO-OP")
      wire#w1
      Contact( #MB3_Decoder.OperationMinus )
      Coil( "A03_HMI".MB3.Button.A0302.Bordatrice.Regolazione.Single_PB[8].Bwd_Minus )
   END_RUNG
   RUNG wire#w1
      Contact( #MB3_Decoder.OperationPlus )
      Coil( "A03_HMI".MB3.Button.A0302.Bordatrice.Regolazione.Single_PB[8].Fwd_Plus )
   END_RUNG
   RUNG wire#w1
      Contact( "A0302_Bordatrice_RegolazioneFormato".AX_M[8].COut.MinusCheckNext )
      Contact( "A03_HMI".MB3.Button.A0302.Bordatrice.Regolazione.Single_PB[8].Bwd_Minus )
      wire#w2
      S_Coil( #MB3_Decoder.OpEnabled )
   END_RUNG
   RUNG wire#w1
      Contact( "A0302_Bordatrice_RegolazioneFormato".AX_M[8].COut.PlusCheckNext )
      Contact( "A03_HMI".MB3.Button.A0302.Bordatrice.Regolazione.Single_PB[8].Fwd_Plus )
   END_RUNG wire#w2
   RUNG wire#w1
      I_Contact( "A0302_Bordatrice_RegolazioneFormato".AX_M[8].COut.Standstill )
      S_Coil( #MB3_Decoder.OpRunning )
   END_RUNG
   RUNG wire#w1
      Contact( "A03_HMI".MB3.Button.A0302.Bordatrice.Regolazione.Single_PB[8].Bwd_Minus )
      Contact( "A0302_Bordatrice_RegolazioneFormato".AX_M[8].COut.MinusLimitReached )
      wire#w3
      S_Coil( #MB3_Decoder.OpDone )
   END_RUNG
   RUNG wire#w1
      Contact( "A03_HMI".MB3.Button.A0302.Bordatrice.Regolazione.Single_PB[8].Fwd_Plus )
      Contact( "A0302_Bordatrice_RegolazioneFormato".AX_M[8].COut.PlusLimitReached )
   END_RUNG wire#w3
   // the same network as SCL:
   #_w1 := #MB3_Decoder.Code = #"4086_BORDATRICE_PASS04_LATO-OP";
   "A03_HMI".MB3.Button.A0302.Bordatrice.Regolazione.Single_PB[8].Bwd_Minus := #_w1 AND #MB3_Decoder.OperationMinus;
   "A03_HMI".MB3.Button.A0302.Bordatrice.Regolazione.Single_PB[8].Fwd_Plus := #_w1 AND #MB3_Decoder.OperationPlus;
   IF #_w1 AND (("A0302_Bordatrice_RegolazioneFormato".AX_M[8].COut.MinusCheckNext AND "A03_HMI".MB3.Button.A0302.Bordatrice.Regolazione.Single_PB[8].Bwd_Minus) OR ("A0302_Bordatrice_RegolazioneFormato".AX_M[8].COut.PlusCheckNext AND "A03_HMI".MB3.Button.A0302.Bordatrice.Regolazione.Single_PB[8].Fwd_Plus)) THEN
       #MB3_Decoder.OpEnabled := TRUE;
   END_IF;
   IF #_w1 AND NOT "A0302_Bordatrice_RegolazioneFormato".AX_M[8].COut.Standstill THEN
       #MB3_Decoder.OpRunning := TRUE;
   END_IF;
   IF #_w1 AND (("A03_HMI".MB3.Button.A0302.Bordatrice.Regolazione.Single_PB[8].Bwd_Minus AND "A0302_Bordatrice_RegolazioneFormato".AX_M[8].COut.MinusLimitReached) OR ("A03_HMI".MB3.Button.A0302.Bordatrice.Regolazione.Single_PB[8].Fwd_Plus AND "A0302_Bordatrice_RegolazioneFormato".AX_M[8].COut.PlusLimitReached)) THEN
       #MB3_Decoder.OpDone := TRUE;
   END_IF;
END_REGION

REGION Network 55: MB3 Code 4098 - REGOLAZ. BORDATRICE - PASSAGGIO 04 - LATO-OP AX-POS
   RUNG wire#powerrail
      { S7_Templates := "SrcType := Int" } EQ_Contact(in1 := #MB3_Decoder.Code, in2 := #"4098_BORDATRICE_PASS04-LATO-OP_AX-POS")
      wire#w1
      { S7_Templates := "SrcType := LReal" } NE_Contact(in1 := "A0302_Bordatrice_RegolazioneFormato".AX_M[8].COut.ActualPosition, in2 := "A0302_Bordatrice_RegolazioneFormato".AX_M[8].HMI.Sts.TargetPos)
      Contact( #MB3_Decoder.OperationPlus )
      Coil( "A03_HMI".MB3.Button.A0302.Bordatrice.Regolazione.Single_PB[8].MoveToPos )
   END_RUNG
   RUNG wire#w1
      Contact( TRUE )
      S_Coil( #MB3_Decoder.OpEnabled )
   END_RUNG
   RUNG wire#w1
      I_Contact( "A0302_Bordatrice_RegolazioneFormato".AX_M[8].COut.Standstill )
      S_Coil( #MB3_Decoder.OpRunning )
   END_RUNG
   RUNG wire#w1
      Contact( "A0302_Bordatrice_RegolazioneFormato".AX_M[8].COut.InPosition )
      S_Coil( #MB3_Decoder.OpDone )
   END_RUNG
   // the same network as SCL:
   #_w1 := #MB3_Decoder.Code = #"4098_BORDATRICE_PASS04-LATO-OP_AX-POS";
   "A03_HMI".MB3.Button.A0302.Bordatrice.Regolazione.Single_PB[8].MoveToPos := #_w1 AND ("A0302_Bordatrice_RegolazioneFormato".AX_M[8].COut.ActualPosition <> "A0302_Bordatrice_RegolazioneFormato".AX_M[8].HMI.Sts.TargetPos) AND #MB3_Decoder.OperationPlus;
   IF #_w1 AND TRUE THEN #MB3_Decoder.OpEnabled := TRUE; END_IF;
   IF #_w1 AND NOT "A0302_Bordatrice_RegolazioneFormato".AX_M[8].COut.Standstill THEN
       #MB3_Decoder.OpRunning := TRUE;
   END_IF;
   IF #_w1 AND "A0302_Bordatrice_RegolazioneFormato".AX_M[8].COut.InPosition THEN
       #MB3_Decoder.OpDone := TRUE;
   END_IF;
END_REGION

REGION Network 56: MB3 Code 4087 - REGOLAZ. BORDATRICE - PASSAGGIO 04 - LATO-MOT
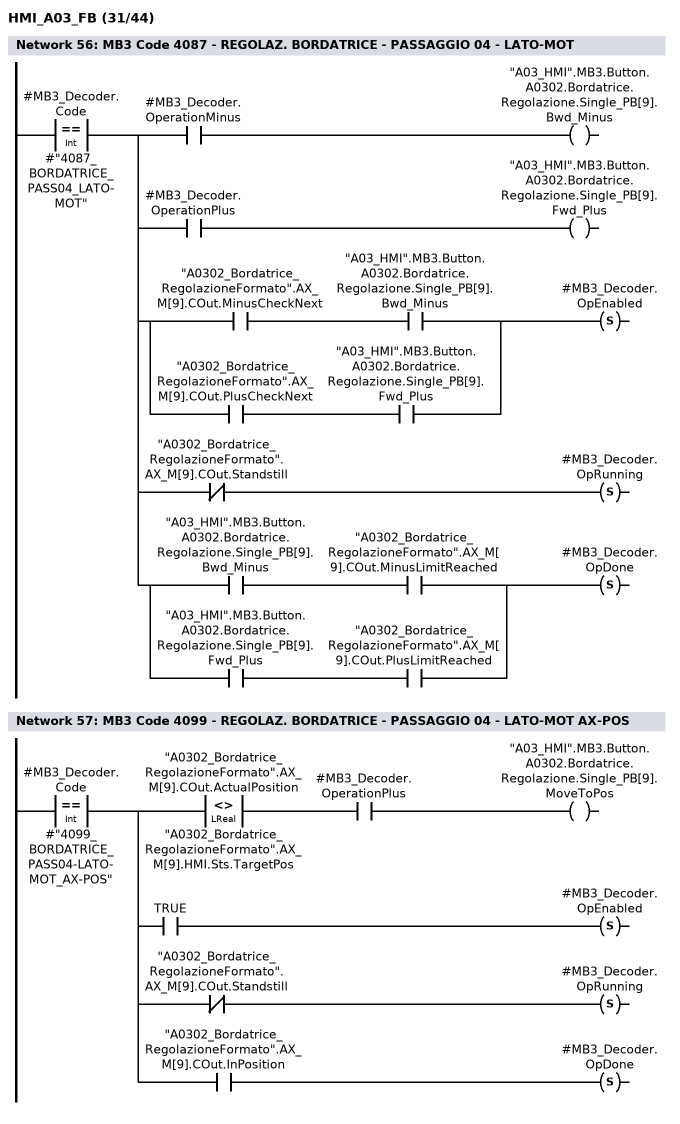
   RUNG wire#powerrail
      { S7_Templates := "SrcType := Int" } EQ_Contact(in1 := #MB3_Decoder.Code, in2 := #"4087_BORDATRICE_PASS04_LATO-MOT")
      wire#w1
      Contact( #MB3_Decoder.OperationMinus )
      Coil( "A03_HMI".MB3.Button.A0302.Bordatrice.Regolazione.Single_PB[9].Bwd_Minus )
   END_RUNG
   RUNG wire#w1
      Contact( #MB3_Decoder.OperationPlus )
      Coil( "A03_HMI".MB3.Button.A0302.Bordatrice.Regolazione.Single_PB[9].Fwd_Plus )
   END_RUNG
   RUNG wire#w1
      Contact( "A0302_Bordatrice_RegolazioneFormato".AX_M[9].COut.MinusCheckNext )
      Contact( "A03_HMI".MB3.Button.A0302.Bordatrice.Regolazione.Single_PB[9].Bwd_Minus )
      wire#w2
      S_Coil( #MB3_Decoder.OpEnabled )
   END_RUNG
   RUNG wire#w1
      Contact( "A0302_Bordatrice_RegolazioneFormato".AX_M[9].COut.PlusCheckNext )
      Contact( "A03_HMI".MB3.Button.A0302.Bordatrice.Regolazione.Single_PB[9].Fwd_Plus )
   END_RUNG wire#w2
   RUNG wire#w1
      I_Contact( "A0302_Bordatrice_RegolazioneFormato".AX_M[9].COut.Standstill )
      S_Coil( #MB3_Decoder.OpRunning )
   END_RUNG
   RUNG wire#w1
      Contact( "A03_HMI".MB3.Button.A0302.Bordatrice.Regolazione.Single_PB[9].Bwd_Minus )
      Contact( "A0302_Bordatrice_RegolazioneFormato".AX_M[9].COut.MinusLimitReached )
      wire#w3
      S_Coil( #MB3_Decoder.OpDone )
   END_RUNG
   RUNG wire#w1
      Contact( "A03_HMI".MB3.Button.A0302.Bordatrice.Regolazione.Single_PB[9].Fwd_Plus )
      Contact( "A0302_Bordatrice_RegolazioneFormato".AX_M[9].COut.PlusLimitReached )
   END_RUNG wire#w3
   // the same network as SCL:
   #_w1 := #MB3_Decoder.Code = #"4087_BORDATRICE_PASS04_LATO-MOT";
   "A03_HMI".MB3.Button.A0302.Bordatrice.Regolazione.Single_PB[9].Bwd_Minus := #_w1 AND #MB3_Decoder.OperationMinus;
   "A03_HMI".MB3.Button.A0302.Bordatrice.Regolazione.Single_PB[9].Fwd_Plus := #_w1 AND #MB3_Decoder.OperationPlus;
   IF #_w1 AND (("A0302_Bordatrice_RegolazioneFormato".AX_M[9].COut.MinusCheckNext AND "A03_HMI".MB3.Button.A0302.Bordatrice.Regolazione.Single_PB[9].Bwd_Minus) OR ("A0302_Bordatrice_RegolazioneFormato".AX_M[9].COut.PlusCheckNext AND "A03_HMI".MB3.Button.A0302.Bordatrice.Regolazione.Single_PB[9].Fwd_Plus)) THEN
       #MB3_Decoder.OpEnabled := TRUE;
   END_IF;
   IF #_w1 AND NOT "A0302_Bordatrice_RegolazioneFormato".AX_M[9].COut.Standstill THEN
       #MB3_Decoder.OpRunning := TRUE;
   END_IF;
   IF #_w1 AND (("A03_HMI".MB3.Button.A0302.Bordatrice.Regolazione.Single_PB[9].Bwd_Minus AND "A0302_Bordatrice_RegolazioneFormato".AX_M[9].COut.MinusLimitReached) OR ("A03_HMI".MB3.Button.A0302.Bordatrice.Regolazione.Single_PB[9].Fwd_Plus AND "A0302_Bordatrice_RegolazioneFormato".AX_M[9].COut.PlusLimitReached)) THEN
       #MB3_Decoder.OpDone := TRUE;
   END_IF;
END_REGION

REGION Network 57: MB3 Code 4099 - REGOLAZ. BORDATRICE - PASSAGGIO 04 - LATO-MOT AX-POS
   RUNG wire#powerrail
      { S7_Templates := "SrcType := Int" } EQ_Contact(in1 := #MB3_Decoder.Code, in2 := #"4099_BORDATRICE_PASS04-LATO-MOT_AX-POS")
      wire#w1
      { S7_Templates := "SrcType := LReal" } NE_Contact(in1 := "A0302_Bordatrice_RegolazioneFormato".AX_M[9].COut.ActualPosition, in2 := "A0302_Bordatrice_RegolazioneFormato".AX_M[9].HMI.Sts.TargetPos)
      Contact( #MB3_Decoder.OperationPlus )
      Coil( "A03_HMI".MB3.Button.A0302.Bordatrice.Regolazione.Single_PB[9].MoveToPos )
   END_RUNG
   RUNG wire#w1
      Contact( TRUE )
      S_Coil( #MB3_Decoder.OpEnabled )
   END_RUNG
   RUNG wire#w1
      I_Contact( "A0302_Bordatrice_RegolazioneFormato".AX_M[9].COut.Standstill )
      S_Coil( #MB3_Decoder.OpRunning )
   END_RUNG
   RUNG wire#w1
      Contact( "A0302_Bordatrice_RegolazioneFormato".AX_M[9].COut.InPosition )
      S_Coil( #MB3_Decoder.OpDone )
   END_RUNG
   // the same network as SCL:
   #_w1 := #MB3_Decoder.Code = #"4099_BORDATRICE_PASS04-LATO-MOT_AX-POS";
   "A03_HMI".MB3.Button.A0302.Bordatrice.Regolazione.Single_PB[9].MoveToPos := #_w1 AND ("A0302_Bordatrice_RegolazioneFormato".AX_M[9].COut.ActualPosition <> "A0302_Bordatrice_RegolazioneFormato".AX_M[9].HMI.Sts.TargetPos) AND #MB3_Decoder.OperationPlus;
   IF #_w1 AND TRUE THEN #MB3_Decoder.OpEnabled := TRUE; END_IF;
   IF #_w1 AND NOT "A0302_Bordatrice_RegolazioneFormato".AX_M[9].COut.Standstill THEN
       #MB3_Decoder.OpRunning := TRUE;
   END_IF;
   IF #_w1 AND "A0302_Bordatrice_RegolazioneFormato".AX_M[9].COut.InPosition THEN
       #MB3_Decoder.OpDone := TRUE;
   END_IF;
END_REGION

REGION Network 58: MB3 Code 4041- CENTARTORI - OP
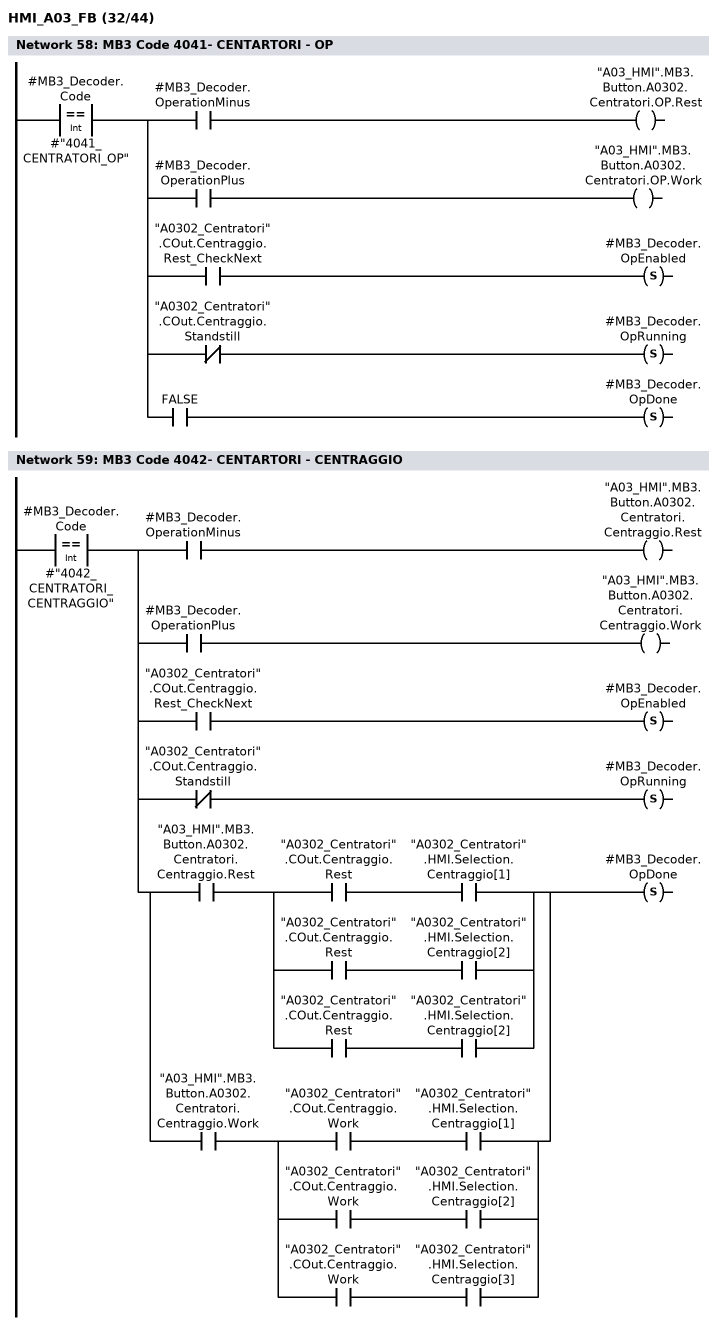
   RUNG wire#powerrail
      { S7_Templates := "SrcType := Int" } EQ_Contact(in1 := #MB3_Decoder.Code, in2 := #"4041_CENTRATORI_OP")
      wire#w1
      Contact( #MB3_Decoder.OperationMinus )
      Coil( "A03_HMI".MB3.Button.A0302.Centratori.OP.Rest )
   END_RUNG
   RUNG wire#w1
      Contact( #MB3_Decoder.OperationPlus )
      Coil( "A03_HMI".MB3.Button.A0302.Centratori.OP.Work )
   END_RUNG
   RUNG wire#w1
      Contact( "A0302_Centratori".COut.Centraggio.Rest_CheckNext )
      S_Coil( #MB3_Decoder.OpEnabled )
   END_RUNG
   RUNG wire#w1
      I_Contact( "A0302_Centratori".COut.Centraggio.Standstill )
      S_Coil( #MB3_Decoder.OpRunning )
   END_RUNG
   RUNG wire#w1
      Contact( FALSE )
      S_Coil( #MB3_Decoder.OpDone )
   END_RUNG
   // the same network as SCL:
   #_w1 := #MB3_Decoder.Code = #"4041_CENTRATORI_OP";
   "A03_HMI".MB3.Button.A0302.Centratori.OP.Rest := #_w1 AND #MB3_Decoder.OperationMinus;
   "A03_HMI".MB3.Button.A0302.Centratori.OP.Work := #_w1 AND #MB3_Decoder.OperationPlus;
   IF #_w1 AND "A0302_Centratori".COut.Centraggio.Rest_CheckNext THEN #MB3_Decoder.OpEnabled := TRUE; END_IF;
   IF #_w1 AND NOT "A0302_Centratori".COut.Centraggio.Standstill THEN #MB3_Decoder.OpRunning := TRUE; END_IF;
   IF #_w1 AND FALSE THEN #MB3_Decoder.OpDone := TRUE; END_IF;
END_REGION

REGION Network 59: MB3 Code 4042- CENTARTORI - CENTRAGGIO
   RUNG wire#powerrail
      { S7_Templates := "SrcType := Int" } EQ_Contact(in1 := #MB3_Decoder.Code, in2 := #"4042_CENTRATORI_CENTRAGGIO")
      wire#w1
      Contact( #MB3_Decoder.OperationMinus )
      Coil( "A03_HMI".MB3.Button.A0302.Centratori.Centraggio.Rest )
   END_RUNG
   RUNG wire#w1
      Contact( #MB3_Decoder.OperationPlus )
      Coil( "A03_HMI".MB3.Button.A0302.Centratori.Centraggio.Work )
   END_RUNG
   RUNG wire#w1
      Contact( "A0302_Centratori".COut.Centraggio.Rest_CheckNext )
      S_Coil( #MB3_Decoder.OpEnabled )
   END_RUNG
   RUNG wire#w1
      I_Contact( "A0302_Centratori".COut.Centraggio.Standstill )
      S_Coil( #MB3_Decoder.OpRunning )
   END_RUNG
   RUNG wire#w1
      Contact( "A03_HMI".MB3.Button.A0302.Centratori.Centraggio.Rest )
      wire#w2
      Contact( "A0302_Centratori".COut.Centraggio.Rest )
      Contact( "A0302_Centratori".HMI.Selection.Centraggio[1] )
      wire#w3
      S_Coil( #MB3_Decoder.OpDone )
   END_RUNG
   RUNG wire#w2
      Contact( "A0302_Centratori".COut.Centraggio.Rest )
      Contact( "A0302_Centratori".HMI.Selection.Centraggio[2] )
   END_RUNG wire#w3
   RUNG wire#w2
      Contact( "A0302_Centratori".COut.Centraggio.Rest )
      Contact( "A0302_Centratori".HMI.Selection.Centraggio[2] )
   END_RUNG wire#w3
   RUNG wire#w1
      Contact( "A03_HMI".MB3.Button.A0302.Centratori.Centraggio.Work )
      wire#w4
      Contact( "A0302_Centratori".COut.Centraggio.Work )
      Contact( "A0302_Centratori".HMI.Selection.Centraggio[1] )
   END_RUNG wire#w3
   RUNG wire#w4
      Contact( "A0302_Centratori".COut.Centraggio.Work )
      Contact( "A0302_Centratori".HMI.Selection.Centraggio[2] )
   END_RUNG wire#w3
   RUNG wire#w4
      Contact( "A0302_Centratori".COut.Centraggio.Work )
      Contact( "A0302_Centratori".HMI.Selection.Centraggio[3] )
   END_RUNG wire#w3
   // the same network as SCL:
   #_w1 := #MB3_Decoder.Code = #"4042_CENTRATORI_CENTRAGGIO";
   "A03_HMI".MB3.Button.A0302.Centratori.Centraggio.Rest := #_w1 AND #MB3_Decoder.OperationMinus;
   "A03_HMI".MB3.Button.A0302.Centratori.Centraggio.Work := #_w1 AND #MB3_Decoder.OperationPlus;
   IF #_w1 AND "A0302_Centratori".COut.Centraggio.Rest_CheckNext THEN #MB3_Decoder.OpEnabled := TRUE; END_IF;
   IF #_w1 AND NOT "A0302_Centratori".COut.Centraggio.Standstill THEN #MB3_Decoder.OpRunning := TRUE; END_IF;
   IF #_w1 AND (("A03_HMI".MB3.Button.A0302.Centratori.Centraggio.Rest AND (("A0302_Centratori".COut.Centraggio.Rest AND "A0302_Centratori".HMI.Selection.Centraggio[1]) OR ("A0302_Centratori".COut.Centraggio.Rest AND "A0302_Centratori".HMI.Selection.Centraggio[2]) OR ("A0302_Centratori".COut.Centraggio.Rest AND "A0302_Centratori".HMI.Selection.Centraggio[2]))) OR ("A03_HMI".MB3.Button.A0302.Centratori.Centraggio.Work AND (("A0302_Centratori".COut.Centraggio.Work AND "A0302_Centratori".HMI.Selection.Centraggio[1]) OR ("A0302_Centratori".COut.Centraggio.Work AND "A0302_Centratori".HMI.Selection.Centraggio[2]) OR ("A0302_Centratori".COut.Centraggio.Work AND "A0302_Centratori".HMI.Selection.Centraggio[3])))) THEN
       #MB3_Decoder.OpDone := TRUE;
   END_IF;
END_REGION

REGION Network 60: MB3 Code 4043- CENTARTORI - SOLLEVAMENTO
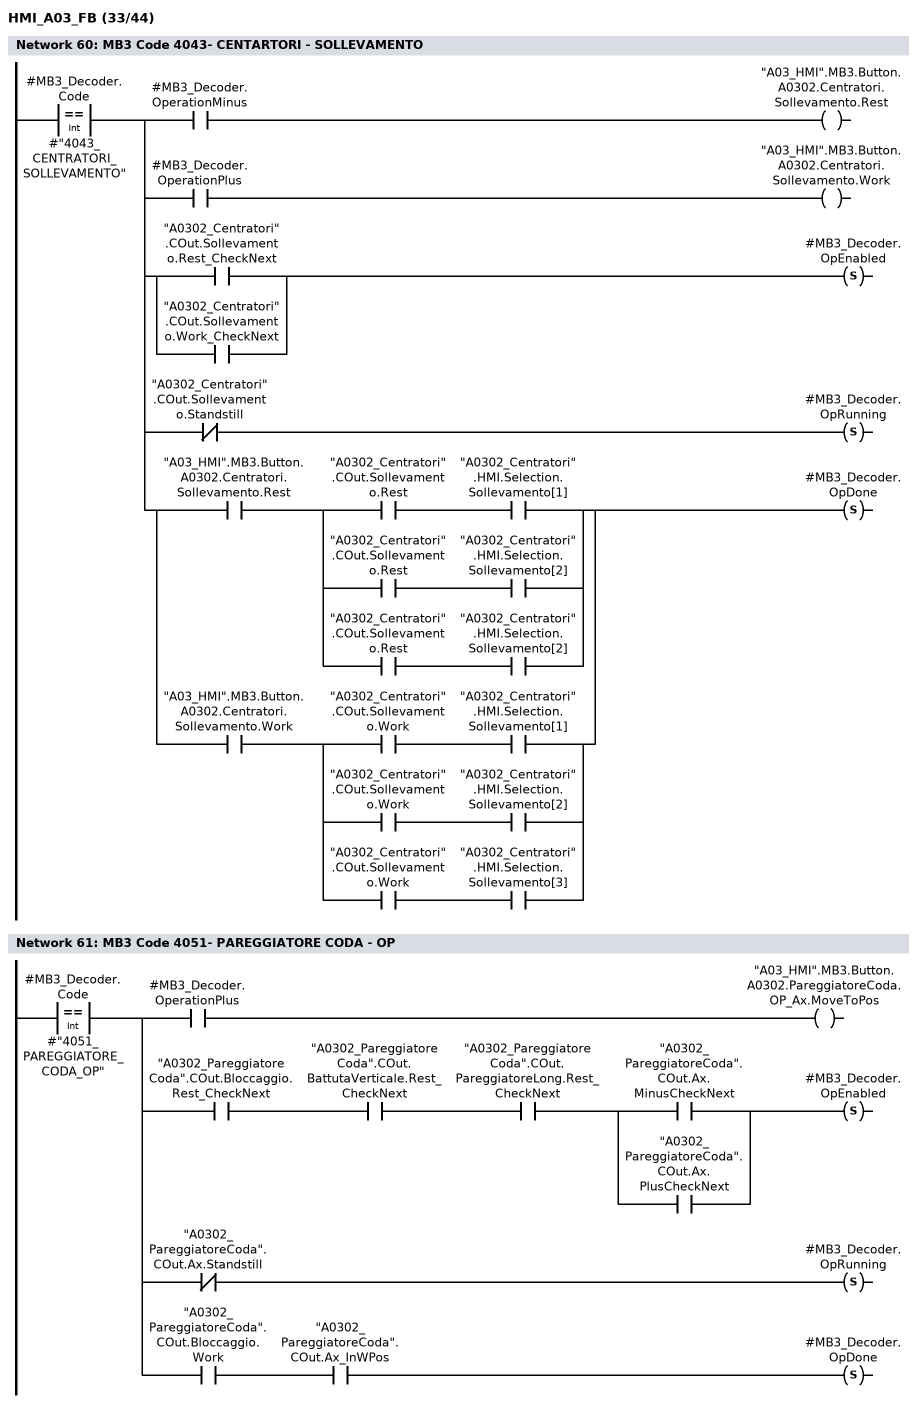
   RUNG wire#powerrail
      { S7_Templates := "SrcType := Int" } EQ_Contact(in1 := #MB3_Decoder.Code, in2 := #"4043_CENTRATORI_SOLLEVAMENTO")
      wire#w1
      Contact( #MB3_Decoder.OperationMinus )
      Coil( "A03_HMI".MB3.Button.A0302.Centratori.Sollevamento.Rest )
   END_RUNG
   RUNG wire#w1
      Contact( #MB3_Decoder.OperationPlus )
      Coil( "A03_HMI".MB3.Button.A0302.Centratori.Sollevamento.Work )
   END_RUNG
   RUNG wire#w1
      Contact( "A0302_Centratori".COut.Sollevamento.Rest_CheckNext )
      wire#w2
      S_Coil( #MB3_Decoder.OpEnabled )
   END_RUNG
   RUNG wire#w1
      Contact( "A0302_Centratori".COut.Sollevamento.Work_CheckNext )
   END_RUNG wire#w2
   RUNG wire#w1
      I_Contact( "A0302_Centratori".COut.Sollevamento.Standstill )
      S_Coil( #MB3_Decoder.OpRunning )
   END_RUNG
   RUNG wire#w1
      Contact( "A03_HMI".MB3.Button.A0302.Centratori.Sollevamento.Rest )
      wire#w3
      Contact( "A0302_Centratori".COut.Sollevamento.Rest )
      Contact( "A0302_Centratori".HMI.Selection.Sollevamento[1] )
      wire#w4
      S_Coil( #MB3_Decoder.OpDone )
   END_RUNG
   RUNG wire#w3
      Contact( "A0302_Centratori".COut.Sollevamento.Rest )
      Contact( "A0302_Centratori".HMI.Selection.Sollevamento[2] )
   END_RUNG wire#w4
   RUNG wire#w3
      Contact( "A0302_Centratori".COut.Sollevamento.Rest )
      Contact( "A0302_Centratori".HMI.Selection.Sollevamento[2] )
   END_RUNG wire#w4
   RUNG wire#w1
      Contact( "A03_HMI".MB3.Button.A0302.Centratori.Sollevamento.Work )
      wire#w5
      Contact( "A0302_Centratori".COut.Sollevamento.Work )
      Contact( "A0302_Centratori".HMI.Selection.Sollevamento[1] )
   END_RUNG wire#w4
   RUNG wire#w5
      Contact( "A0302_Centratori".COut.Sollevamento.Work )
      Contact( "A0302_Centratori".HMI.Selection.Sollevamento[2] )
   END_RUNG wire#w4
   RUNG wire#w5
      Contact( "A0302_Centratori".COut.Sollevamento.Work )
      Contact( "A0302_Centratori".HMI.Selection.Sollevamento[3] )
   END_RUNG wire#w4
   // the same network as SCL:
   #_w1 := #MB3_Decoder.Code = #"4043_CENTRATORI_SOLLEVAMENTO";
   "A03_HMI".MB3.Button.A0302.Centratori.Sollevamento.Rest := #_w1 AND #MB3_Decoder.OperationMinus;
   "A03_HMI".MB3.Button.A0302.Centratori.Sollevamento.Work := #_w1 AND #MB3_Decoder.OperationPlus;
   IF #_w1 AND ("A0302_Centratori".COut.Sollevamento.Rest_CheckNext OR "A0302_Centratori".COut.Sollevamento.Work_CheckNext) THEN
       #MB3_Decoder.OpEnabled := TRUE;
   END_IF;
   IF #_w1 AND NOT "A0302_Centratori".COut.Sollevamento.Standstill THEN
       #MB3_Decoder.OpRunning := TRUE;
   END_IF;
   IF #_w1 AND (("A03_HMI".MB3.Button.A0302.Centratori.Sollevamento.Rest AND (("A0302_Centratori".COut.Sollevamento.Rest AND "A0302_Centratori".HMI.Selection.Sollevamento[1]) OR ("A0302_Centratori".COut.Sollevamento.Rest AND "A0302_Centratori".HMI.Selection.Sollevamento[2]) OR ("A0302_Centratori".COut.Sollevamento.Rest AND "A0302_Centratori".HMI.Selection.Sollevamento[2]))) OR ("A03_HMI".MB3.Button.A0302.Centratori.Sollevamento.Work AND (("A0302_Centratori".COut.Sollevamento.Work AND "A0302_Centratori".HMI.Selection.Sollevamento[1]) OR ("A0302_Centratori".COut.Sollevamento.Work AND "A0302_Centratori".HMI.Selection.Sollevamento[2]) OR ("A0302_Centratori".COut.Sollevamento.Work AND "A0302_Centratori".HMI.Selection.Sollevamento[3])))) THEN
       #MB3_Decoder.OpDone := TRUE;
   END_IF;
END_REGION

REGION Network 61: MB3 Code 4051- PAREGGIATORE CODA - OP
   RUNG wire#powerrail
      { S7_Templates := "SrcType := Int" } EQ_Contact(in1 := #MB3_Decoder.Code, in2 := #"4051_PAREGGIATORE_CODA_OP")
      wire#w1
      Contact( #MB3_Decoder.OperationPlus )
      Coil( "A03_HMI".MB3.Button.A0302.PareggiatoreCoda.OP_Ax.MoveToPos )
   END_RUNG
   RUNG wire#w1
      Contact( "A0302_PareggiatoreCoda".COut.Bloccaggio.Rest_CheckNext )
      Contact( "A0302_PareggiatoreCoda".COut.BattutaVerticale.Rest_CheckNext )
      Contact( "A0302_PareggiatoreCoda".COut.PareggiatoreLong.Rest_CheckNext )
      wire#w2
      Contact( "A0302_PareggiatoreCoda".COut.Ax.MinusCheckNext )
      wire#w3
      S_Coil( #MB3_Decoder.OpEnabled )
   END_RUNG
   RUNG wire#w2
      Contact( "A0302_PareggiatoreCoda".COut.Ax.PlusCheckNext )
   END_RUNG wire#w3
   RUNG wire#w1
      I_Contact( "A0302_PareggiatoreCoda".COut.Ax.Standstill )
      S_Coil( #MB3_Decoder.OpRunning )
   END_RUNG
   RUNG wire#w1
      Contact( "A0302_PareggiatoreCoda".COut.Bloccaggio.Work )
      Contact( "A0302_PareggiatoreCoda".COut.Ax_InWPos )
      S_Coil( #MB3_Decoder.OpDone )
   END_RUNG
   // the same network as SCL:
   #_w1 := #MB3_Decoder.Code = #"4051_PAREGGIATORE_CODA_OP";
   "A03_HMI".MB3.Button.A0302.PareggiatoreCoda.OP_Ax.MoveToPos := #_w1 AND #MB3_Decoder.OperationPlus;
   IF #_w1 AND "A0302_PareggiatoreCoda".COut.Bloccaggio.Rest_CheckNext AND "A0302_PareggiatoreCoda".COut.BattutaVerticale.Rest_CheckNext AND "A0302_PareggiatoreCoda".COut.PareggiatoreLong.Rest_CheckNext AND ("A0302_PareggiatoreCoda".COut.Ax.MinusCheckNext OR "A0302_PareggiatoreCoda".COut.Ax.PlusCheckNext) THEN
       #MB3_Decoder.OpEnabled := TRUE;
   END_IF;
   IF #_w1 AND NOT "A0302_PareggiatoreCoda".COut.Ax.Standstill THEN #MB3_Decoder.OpRunning := TRUE; END_IF;
   IF #_w1 AND "A0302_PareggiatoreCoda".COut.Bloccaggio.Work AND "A0302_PareggiatoreCoda".COut.Ax_InWPos THEN
       #MB3_Decoder.OpDone := TRUE;
   END_IF;
END_REGION

REGION Network 62: MB3 Code 4052 - PAREGGIATORE CODA -AX
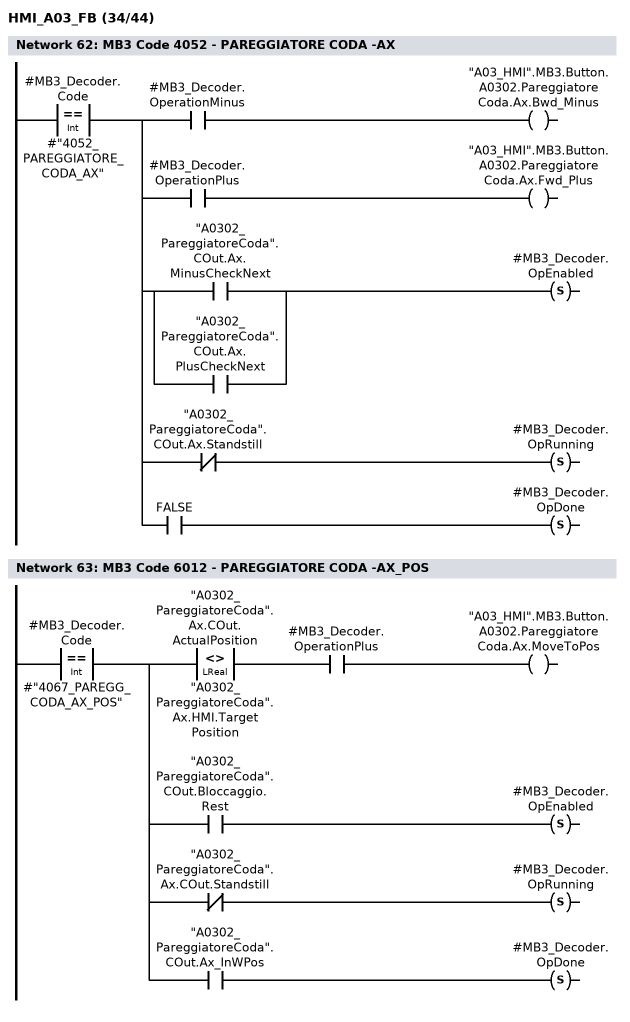
   RUNG wire#powerrail
      { S7_Templates := "SrcType := Int" } EQ_Contact(in1 := #MB3_Decoder.Code, in2 := #"4052_PAREGGIATORE_CODA_AX")
      wire#w1
      Contact( #MB3_Decoder.OperationMinus )
      Coil( "A03_HMI".MB3.Button.A0302.PareggiatoreCoda.Ax.Bwd_Minus )
   END_RUNG
   RUNG wire#w1
      Contact( #MB3_Decoder.OperationPlus )
      Coil( "A03_HMI".MB3.Button.A0302.PareggiatoreCoda.Ax.Fwd_Plus )
   END_RUNG
   RUNG wire#w1
      Contact( "A0302_PareggiatoreCoda".COut.Ax.MinusCheckNext )
      wire#w2
      S_Coil( #MB3_Decoder.OpEnabled )
   END_RUNG
   RUNG wire#w1
      Contact( "A0302_PareggiatoreCoda".COut.Ax.PlusCheckNext )
   END_RUNG wire#w2
   RUNG wire#w1
      I_Contact( "A0302_PareggiatoreCoda".COut.Ax.Standstill )
      S_Coil( #MB3_Decoder.OpRunning )
   END_RUNG
   RUNG wire#w1
      Contact( FALSE )
      S_Coil( #MB3_Decoder.OpDone )
   END_RUNG
   // the same network as SCL:
   #_w1 := #MB3_Decoder.Code = #"4052_PAREGGIATORE_CODA_AX";
   "A03_HMI".MB3.Button.A0302.PareggiatoreCoda.Ax.Bwd_Minus := #_w1 AND #MB3_Decoder.OperationMinus;
   "A03_HMI".MB3.Button.A0302.PareggiatoreCoda.Ax.Fwd_Plus := #_w1 AND #MB3_Decoder.OperationPlus;
   IF #_w1 AND ("A0302_PareggiatoreCoda".COut.Ax.MinusCheckNext OR "A0302_PareggiatoreCoda".COut.Ax.PlusCheckNext) THEN
       #MB3_Decoder.OpEnabled := TRUE;
   END_IF;
   IF #_w1 AND NOT "A0302_PareggiatoreCoda".COut.Ax.Standstill THEN #MB3_Decoder.OpRunning := TRUE; END_IF;
   IF #_w1 AND FALSE THEN #MB3_Decoder.OpDone := TRUE; END_IF;
END_REGION

REGION Network 63: MB3 Code 6012 - PAREGGIATORE CODA -AX_POS
   RUNG wire#powerrail
      { S7_Templates := "SrcType := Int" } EQ_Contact(in1 := #MB3_Decoder.Code, in2 := #"4067_PAREGG_CODA_AX_POS")
      wire#w1
      { S7_Templates := "SrcType := LReal" } NE_Contact(in1 := "A0302_PareggiatoreCoda".Ax.COut.ActualPosition, in2 := "A0302_PareggiatoreCoda".Ax.HMI.TargetPosition)
      Contact( #MB3_Decoder.OperationPlus )
      Coil( "A03_HMI".MB3.Button.A0302.PareggiatoreCoda.Ax.MoveToPos )
   END_RUNG
   RUNG wire#w1
      Contact( "A0302_PareggiatoreCoda".COut.Bloccaggio.Rest )
      S_Coil( #MB3_Decoder.OpEnabled )
   END_RUNG
   RUNG wire#w1
      I_Contact( "A0302_PareggiatoreCoda".Ax.COut.Standstill )
      S_Coil( #MB3_Decoder.OpRunning )
   END_RUNG
   RUNG wire#w1
      Contact( "A0302_PareggiatoreCoda".COut.Ax_InWPos )
      S_Coil( #MB3_Decoder.OpDone )
   END_RUNG
   // the same network as SCL:
   #_w1 := #MB3_Decoder.Code = #"4067_PAREGG_CODA_AX_POS";
   "A03_HMI".MB3.Button.A0302.PareggiatoreCoda.Ax.MoveToPos := #_w1 AND ("A0302_PareggiatoreCoda".Ax.COut.ActualPosition <> "A0302_PareggiatoreCoda".Ax.HMI.TargetPosition) AND #MB3_Decoder.OperationPlus;
   IF #_w1 AND "A0302_PareggiatoreCoda".COut.Bloccaggio.Rest THEN #MB3_Decoder.OpEnabled := TRUE; END_IF;
   IF #_w1 AND NOT "A0302_PareggiatoreCoda".Ax.COut.Standstill THEN #MB3_Decoder.OpRunning := TRUE; END_IF;
   IF #_w1 AND "A0302_PareggiatoreCoda".COut.Ax_InWPos THEN #MB3_Decoder.OpDone := TRUE; END_IF;
END_REGION

REGION Network 64: MB3 Code 4053 - PAREGGIATORE CODA - BLOCCAGGIO
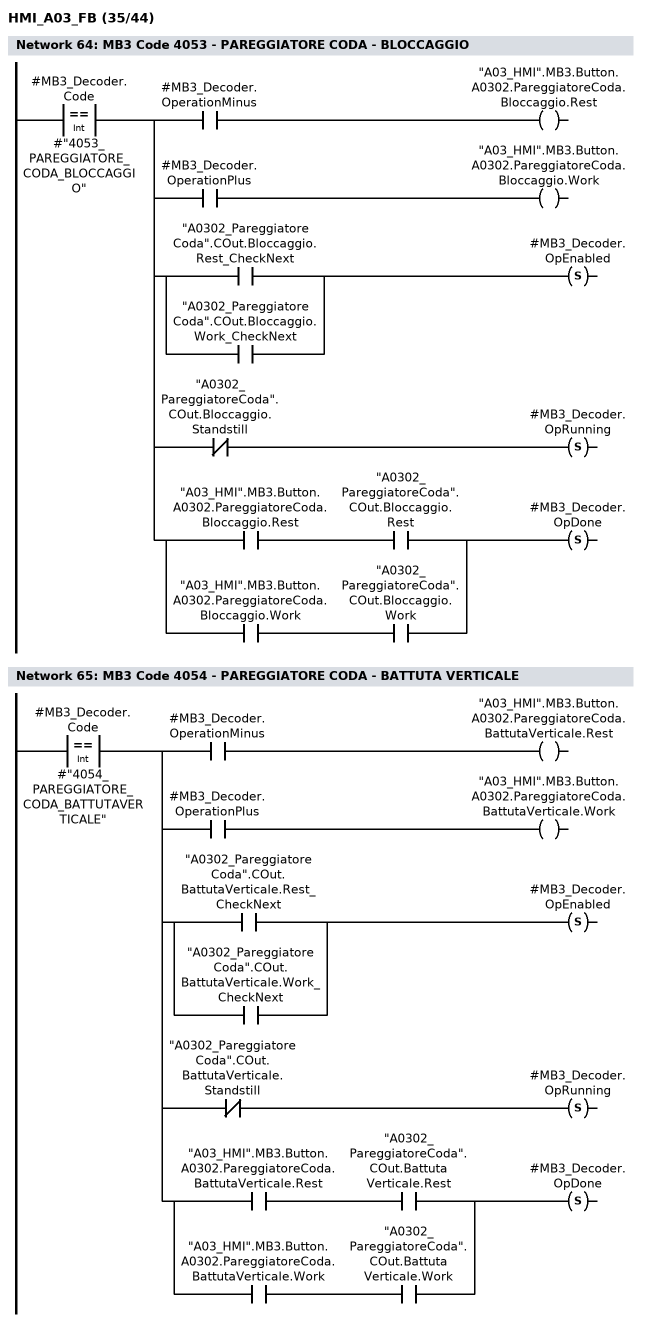
   RUNG wire#powerrail
      { S7_Templates := "SrcType := Int" } EQ_Contact(in1 := #MB3_Decoder.Code, in2 := #"4053_PAREGGIATORE_CODA_BLOCCAGGIO")
      wire#w1
      Contact( #MB3_Decoder.OperationMinus )
      Coil( "A03_HMI".MB3.Button.A0302.PareggiatoreCoda.Bloccaggio.Rest )
   END_RUNG
   RUNG wire#w1
      Contact( #MB3_Decoder.OperationPlus )
      Coil( "A03_HMI".MB3.Button.A0302.PareggiatoreCoda.Bloccaggio.Work )
   END_RUNG
   RUNG wire#w1
      Contact( "A0302_PareggiatoreCoda".COut.Bloccaggio.Rest_CheckNext )
      wire#w2
      S_Coil( #MB3_Decoder.OpEnabled )
   END_RUNG
   RUNG wire#w1
      Contact( "A0302_PareggiatoreCoda".COut.Bloccaggio.Work_CheckNext )
   END_RUNG wire#w2
   RUNG wire#w1
      I_Contact( "A0302_PareggiatoreCoda".COut.Bloccaggio.Standstill )
      S_Coil( #MB3_Decoder.OpRunning )
   END_RUNG
   RUNG wire#w1
      Contact( "A03_HMI".MB3.Button.A0302.PareggiatoreCoda.Bloccaggio.Rest )
      Contact( "A0302_PareggiatoreCoda".COut.Bloccaggio.Rest )
      wire#w3
      S_Coil( #MB3_Decoder.OpDone )
   END_RUNG
   RUNG wire#w1
      Contact( "A03_HMI".MB3.Button.A0302.PareggiatoreCoda.Bloccaggio.Work )
      Contact( "A0302_PareggiatoreCoda".COut.Bloccaggio.Work )
   END_RUNG wire#w3
   // the same network as SCL:
   #_w1 := #MB3_Decoder.Code = #"4053_PAREGGIATORE_CODA_BLOCCAGGIO";
   "A03_HMI".MB3.Button.A0302.PareggiatoreCoda.Bloccaggio.Rest := #_w1 AND #MB3_Decoder.OperationMinus;
   "A03_HMI".MB3.Button.A0302.PareggiatoreCoda.Bloccaggio.Work := #_w1 AND #MB3_Decoder.OperationPlus;
   IF #_w1 AND ("A0302_PareggiatoreCoda".COut.Bloccaggio.Rest_CheckNext OR "A0302_PareggiatoreCoda".COut.Bloccaggio.Work_CheckNext) THEN
       #MB3_Decoder.OpEnabled := TRUE;
   END_IF;
   IF #_w1 AND NOT "A0302_PareggiatoreCoda".COut.Bloccaggio.Standstill THEN
       #MB3_Decoder.OpRunning := TRUE;
   END_IF;
   IF #_w1 AND (("A03_HMI".MB3.Button.A0302.PareggiatoreCoda.Bloccaggio.Rest AND "A0302_PareggiatoreCoda".COut.Bloccaggio.Rest) OR ("A03_HMI".MB3.Button.A0302.PareggiatoreCoda.Bloccaggio.Work AND "A0302_PareggiatoreCoda".COut.Bloccaggio.Work)) THEN
       #MB3_Decoder.OpDone := TRUE;
   END_IF;
END_REGION

REGION Network 65: MB3 Code 4054 - PAREGGIATORE CODA - BATTUTA VERTICALE
   RUNG wire#powerrail
      { S7_Templates := "SrcType := Int" } EQ_Contact(in1 := #MB3_Decoder.Code, in2 := #"4054_PAREGGIATORE_CODA_BATTUTAVERTICALE")
      wire#w1
      Contact( #MB3_Decoder.OperationMinus )
      Coil( "A03_HMI".MB3.Button.A0302.PareggiatoreCoda.BattutaVerticale.Rest )
   END_RUNG
   RUNG wire#w1
      Contact( #MB3_Decoder.OperationPlus )
      Coil( "A03_HMI".MB3.Button.A0302.PareggiatoreCoda.BattutaVerticale.Work )
   END_RUNG
   RUNG wire#w1
      Contact( "A0302_PareggiatoreCoda".COut.BattutaVerticale.Rest_CheckNext )
      wire#w2
      S_Coil( #MB3_Decoder.OpEnabled )
   END_RUNG
   RUNG wire#w1
      Contact( "A0302_PareggiatoreCoda".COut.BattutaVerticale.Work_CheckNext )
   END_RUNG wire#w2
   RUNG wire#w1
      I_Contact( "A0302_PareggiatoreCoda".COut.BattutaVerticale.Standstill )
      S_Coil( #MB3_Decoder.OpRunning )
   END_RUNG
   RUNG wire#w1
      Contact( "A03_HMI".MB3.Button.A0302.PareggiatoreCoda.BattutaVerticale.Rest )
      Contact( "A0302_PareggiatoreCoda".COut.BattutaVerticale.Rest )
      wire#w3
      S_Coil( #MB3_Decoder.OpDone )
   END_RUNG
   RUNG wire#w1
      Contact( "A03_HMI".MB3.Button.A0302.PareggiatoreCoda.BattutaVerticale.Work )
      Contact( "A0302_PareggiatoreCoda".COut.BattutaVerticale.Work )
   END_RUNG wire#w3
   // the same network as SCL:
   #_w1 := #MB3_Decoder.Code = #"4054_PAREGGIATORE_CODA_BATTUTAVERTICALE";
   "A03_HMI".MB3.Button.A0302.PareggiatoreCoda.BattutaVerticale.Rest := #_w1 AND #MB3_Decoder.OperationMinus;
   "A03_HMI".MB3.Button.A0302.PareggiatoreCoda.BattutaVerticale.Work := #_w1 AND #MB3_Decoder.OperationPlus;
   IF #_w1 AND ("A0302_PareggiatoreCoda".COut.BattutaVerticale.Rest_CheckNext OR "A0302_PareggiatoreCoda".COut.BattutaVerticale.Work_CheckNext) THEN
       #MB3_Decoder.OpEnabled := TRUE;
   END_IF;
   IF #_w1 AND NOT "A0302_PareggiatoreCoda".COut.BattutaVerticale.Standstill THEN
       #MB3_Decoder.OpRunning := TRUE;
   END_IF;
   IF #_w1 AND (("A03_HMI".MB3.Button.A0302.PareggiatoreCoda.BattutaVerticale.Rest AND "A0302_PareggiatoreCoda".COut.BattutaVerticale.Rest) OR ("A03_HMI".MB3.Button.A0302.PareggiatoreCoda.BattutaVerticale.Work AND "A0302_PareggiatoreCoda".COut.BattutaVerticale.Work)) THEN
       #MB3_Decoder.OpDone := TRUE;
   END_IF;
END_REGION

REGION Network 66: MB3 Code 4055 - PAREGGIATORE CODA - PAREGGIATORE LONGITUDINALE
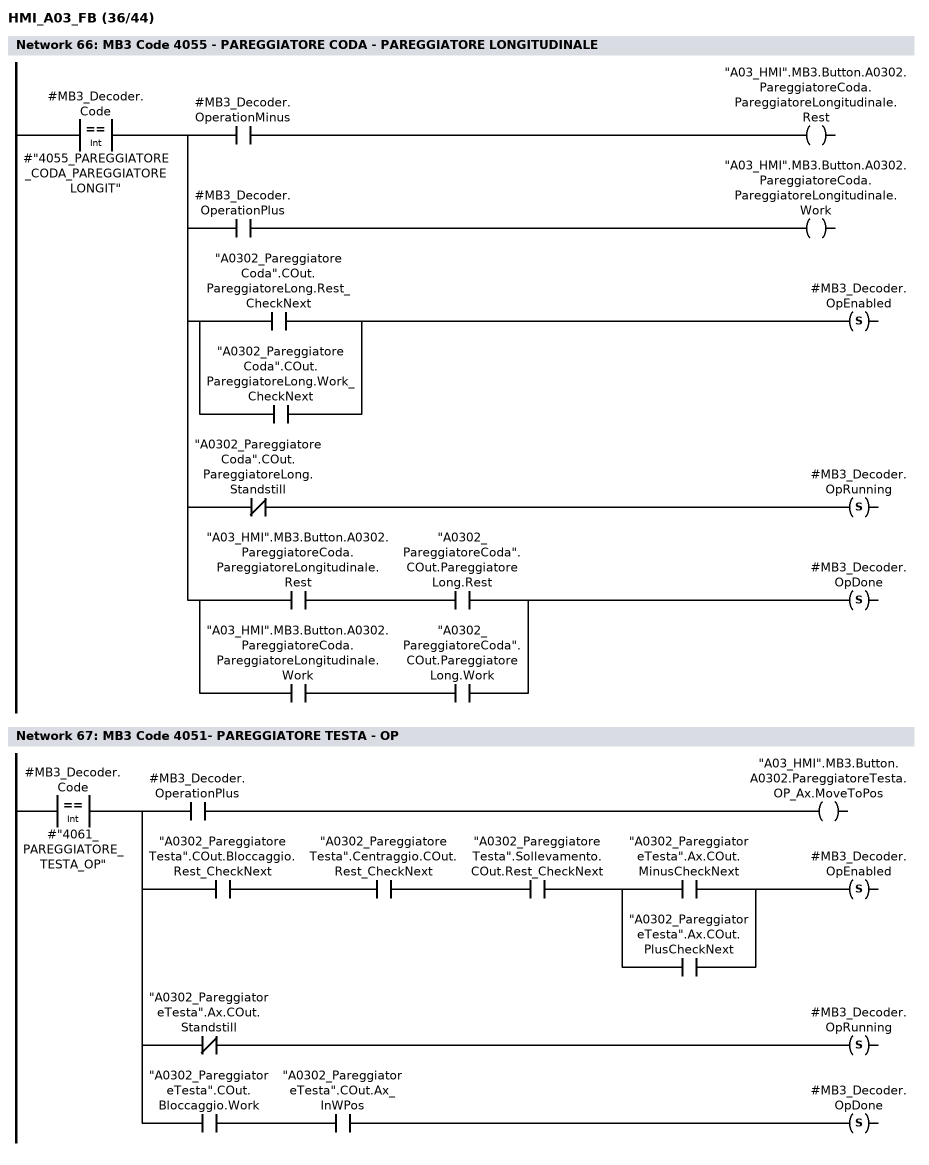
   RUNG wire#powerrail
      { S7_Templates := "SrcType := Int" } EQ_Contact(in1 := #MB3_Decoder.Code, in2 := #"4055_PAREGGIATORE_CODA_PAREGGIATORELONGIT")
      wire#w1
      Contact( #MB3_Decoder.OperationMinus )
      Coil( "A03_HMI".MB3.Button.A0302.PareggiatoreCoda.PareggiatoreLongitudinale.Rest )
   END_RUNG
   RUNG wire#w1
      Contact( #MB3_Decoder.OperationPlus )
      Coil( "A03_HMI".MB3.Button.A0302.PareggiatoreCoda.PareggiatoreLongitudinale.Work )
   END_RUNG
   RUNG wire#w1
      Contact( "A0302_PareggiatoreCoda".COut.PareggiatoreLong.Rest_CheckNext )
      wire#w2
      S_Coil( #MB3_Decoder.OpEnabled )
   END_RUNG
   RUNG wire#w1
      Contact( "A0302_PareggiatoreCoda".COut.PareggiatoreLong.Work_CheckNext )
   END_RUNG wire#w2
   RUNG wire#w1
      I_Contact( "A0302_PareggiatoreCoda".COut.PareggiatoreLong.Standstill )
      S_Coil( #MB3_Decoder.OpRunning )
   END_RUNG
   RUNG wire#w1
      Contact( "A03_HMI".MB3.Button.A0302.PareggiatoreCoda.PareggiatoreLongitudinale.Rest )
      Contact( "A0302_PareggiatoreCoda".COut.PareggiatoreLong.Rest )
      wire#w3
      S_Coil( #MB3_Decoder.OpDone )
   END_RUNG
   RUNG wire#w1
      Contact( "A03_HMI".MB3.Button.A0302.PareggiatoreCoda.PareggiatoreLongitudinale.Work )
      Contact( "A0302_PareggiatoreCoda".COut.PareggiatoreLong.Work )
   END_RUNG wire#w3
   // the same network as SCL:
   #_w1 := #MB3_Decoder.Code = #"4055_PAREGGIATORE_CODA_PAREGGIATORELONGIT";
   "A03_HMI".MB3.Button.A0302.PareggiatoreCoda.PareggiatoreLongitudinale.Rest := #_w1 AND #MB3_Decoder.OperationMinus;
   "A03_HMI".MB3.Button.A0302.PareggiatoreCoda.PareggiatoreLongitudinale.Work := #_w1 AND #MB3_Decoder.OperationPlus;
   IF #_w1 AND ("A0302_PareggiatoreCoda".COut.PareggiatoreLong.Rest_CheckNext OR "A0302_PareggiatoreCoda".COut.PareggiatoreLong.Work_CheckNext) THEN
       #MB3_Decoder.OpEnabled := TRUE;
   END_IF;
   IF #_w1 AND NOT "A0302_PareggiatoreCoda".COut.PareggiatoreLong.Standstill THEN
       #MB3_Decoder.OpRunning := TRUE;
   END_IF;
   IF #_w1 AND (("A03_HMI".MB3.Button.A0302.PareggiatoreCoda.PareggiatoreLongitudinale.Rest AND "A0302_PareggiatoreCoda".COut.PareggiatoreLong.Rest) OR ("A03_HMI".MB3.Button.A0302.PareggiatoreCoda.PareggiatoreLongitudinale.Work AND "A0302_PareggiatoreCoda".COut.PareggiatoreLong.Work)) THEN
       #MB3_Decoder.OpDone := TRUE;
   END_IF;
END_REGION

REGION Network 67: MB3 Code 4051- PAREGGIATORE TESTA - OP
   RUNG wire#powerrail
      { S7_Templates := "SrcType := Int" } EQ_Contact(in1 := #MB3_Decoder.Code, in2 := #"4061_PAREGGIATORE_TESTA_OP")
      wire#w1
      Contact( #MB3_Decoder.OperationPlus )
      Coil( "A03_HMI".MB3.Button.A0302.PareggiatoreTesta.OP_Ax.MoveToPos )
   END_RUNG
   RUNG wire#w1
      Contact( "A0302_PareggiatoreTesta".COut.Bloccaggio.Rest_CheckNext )
      Contact( "A0302_PareggiatoreTesta".Centraggio.COut.Rest_CheckNext )
      Contact( "A0302_PareggiatoreTesta".Sollevamento.COut.Rest_CheckNext )
      wire#w2
      Contact( "A0302_PareggiatoreTesta".Ax.COut.MinusCheckNext )
      wire#w3
      S_Coil( #MB3_Decoder.OpEnabled )
   END_RUNG
   RUNG wire#w2
      Contact( "A0302_PareggiatoreTesta".Ax.COut.PlusCheckNext )
   END_RUNG wire#w3
   RUNG wire#w1
      I_Contact( "A0302_PareggiatoreTesta".Ax.COut.Standstill )
      S_Coil( #MB3_Decoder.OpRunning )
   END_RUNG
   RUNG wire#w1
      Contact( "A0302_PareggiatoreTesta".COut.Bloccaggio.Work )
      Contact( "A0302_PareggiatoreTesta".COut.Ax_InWPos )
      S_Coil( #MB3_Decoder.OpDone )
   END_RUNG
   // the same network as SCL:
   #_w1 := #MB3_Decoder.Code = #"4061_PAREGGIATORE_TESTA_OP";
   "A03_HMI".MB3.Button.A0302.PareggiatoreTesta.OP_Ax.MoveToPos := #_w1 AND #MB3_Decoder.OperationPlus;
   IF #_w1 AND "A0302_PareggiatoreTesta".COut.Bloccaggio.Rest_CheckNext AND "A0302_PareggiatoreTesta".Centraggio.COut.Rest_CheckNext AND "A0302_PareggiatoreTesta".Sollevamento.COut.Rest_CheckNext AND ("A0302_PareggiatoreTesta".Ax.COut.MinusCheckNext OR "A0302_PareggiatoreTesta".Ax.COut.PlusCheckNext) THEN
       #MB3_Decoder.OpEnabled := TRUE;
   END_IF;
   IF #_w1 AND NOT "A0302_PareggiatoreTesta".Ax.COut.Standstill THEN #MB3_Decoder.OpRunning := TRUE; END_IF;
   IF #_w1 AND "A0302_PareggiatoreTesta".COut.Bloccaggio.Work AND "A0302_PareggiatoreTesta".COut.Ax_InWPos THEN
       #MB3_Decoder.OpDone := TRUE;
   END_IF;
END_REGION

REGION Network 68: MB3 Code 4062 - PAREGGIATORE TESTA -AX
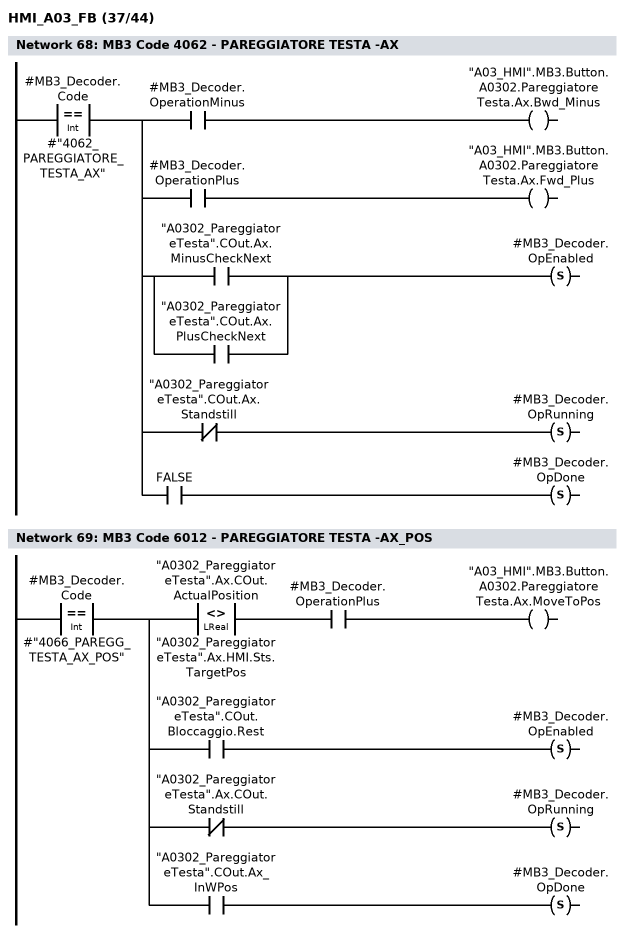
   RUNG wire#powerrail
      { S7_Templates := "SrcType := Int" } EQ_Contact(in1 := #MB3_Decoder.Code, in2 := #"4062_PAREGGIATORE_TESTA_AX")
      wire#w1
      Contact( #MB3_Decoder.OperationMinus )
      Coil( "A03_HMI".MB3.Button.A0302.PareggiatoreTesta.Ax.Bwd_Minus )
   END_RUNG
   RUNG wire#w1
      Contact( #MB3_Decoder.OperationPlus )
      Coil( "A03_HMI".MB3.Button.A0302.PareggiatoreTesta.Ax.Fwd_Plus )
   END_RUNG
   RUNG wire#w1
      Contact( "A0302_PareggiatoreTesta".COut.Ax.MinusCheckNext )
      wire#w2
      S_Coil( #MB3_Decoder.OpEnabled )
   END_RUNG
   RUNG wire#w1
      Contact( "A0302_PareggiatoreTesta".COut.Ax.PlusCheckNext )
   END_RUNG wire#w2
   RUNG wire#w1
      I_Contact( "A0302_PareggiatoreTesta".COut.Ax.Standstill )
      S_Coil( #MB3_Decoder.OpRunning )
   END_RUNG
   RUNG wire#w1
      Contact( FALSE )
      S_Coil( #MB3_Decoder.OpDone )
   END_RUNG
   // the same network as SCL:
   #_w1 := #MB3_Decoder.Code = #"4062_PAREGGIATORE_TESTA_AX";
   "A03_HMI".MB3.Button.A0302.PareggiatoreTesta.Ax.Bwd_Minus := #_w1 AND #MB3_Decoder.OperationMinus;
   "A03_HMI".MB3.Button.A0302.PareggiatoreTesta.Ax.Fwd_Plus := #_w1 AND #MB3_Decoder.OperationPlus;
   IF #_w1 AND ("A0302_PareggiatoreTesta".COut.Ax.MinusCheckNext OR "A0302_PareggiatoreTesta".COut.Ax.PlusCheckNext) THEN
       #MB3_Decoder.OpEnabled := TRUE;
   END_IF;
   IF #_w1 AND NOT "A0302_PareggiatoreTesta".COut.Ax.Standstill THEN #MB3_Decoder.OpRunning := TRUE; END_IF;
   IF #_w1 AND FALSE THEN #MB3_Decoder.OpDone := TRUE; END_IF;
END_REGION

REGION Network 69: MB3 Code 6012 - PAREGGIATORE TESTA -AX_POS
   RUNG wire#powerrail
      { S7_Templates := "SrcType := Int" } EQ_Contact(in1 := #MB3_Decoder.Code, in2 := #"4066_PAREGG_TESTA_AX_POS")
      wire#w1
      { S7_Templates := "SrcType := LReal" } NE_Contact(in1 := "A0302_PareggiatoreTesta".Ax.COut.ActualPosition, in2 := "A0302_PareggiatoreTesta".Ax.HMI.Sts.TargetPos)
      Contact( #MB3_Decoder.OperationPlus )
      Coil( "A03_HMI".MB3.Button.A0302.PareggiatoreTesta.Ax.MoveToPos )
   END_RUNG
   RUNG wire#w1
      Contact( "A0302_PareggiatoreTesta".COut.Bloccaggio.Rest )
      S_Coil( #MB3_Decoder.OpEnabled )
   END_RUNG
   RUNG wire#w1
      I_Contact( "A0302_PareggiatoreTesta".Ax.COut.Standstill )
      S_Coil( #MB3_Decoder.OpRunning )
   END_RUNG
   RUNG wire#w1
      Contact( "A0302_PareggiatoreTesta".COut.Ax_InWPos )
      S_Coil( #MB3_Decoder.OpDone )
   END_RUNG
   // the same network as SCL:
   #_w1 := #MB3_Decoder.Code = #"4066_PAREGG_TESTA_AX_POS";
   "A03_HMI".MB3.Button.A0302.PareggiatoreTesta.Ax.MoveToPos := #_w1 AND ("A0302_PareggiatoreTesta".Ax.COut.ActualPosition <> "A0302_PareggiatoreTesta".Ax.HMI.Sts.TargetPos) AND #MB3_Decoder.OperationPlus;
   IF #_w1 AND "A0302_PareggiatoreTesta".COut.Bloccaggio.Rest THEN #MB3_Decoder.OpEnabled := TRUE; END_IF;
   IF #_w1 AND NOT "A0302_PareggiatoreTesta".Ax.COut.Standstill THEN #MB3_Decoder.OpRunning := TRUE; END_IF;
   IF #_w1 AND "A0302_PareggiatoreTesta".COut.Ax_InWPos THEN #MB3_Decoder.OpDone := TRUE; END_IF;
END_REGION

REGION Network 70: MB3 Code 4063 - PAREGGIATORE TESTA - BLOCCAGGIO
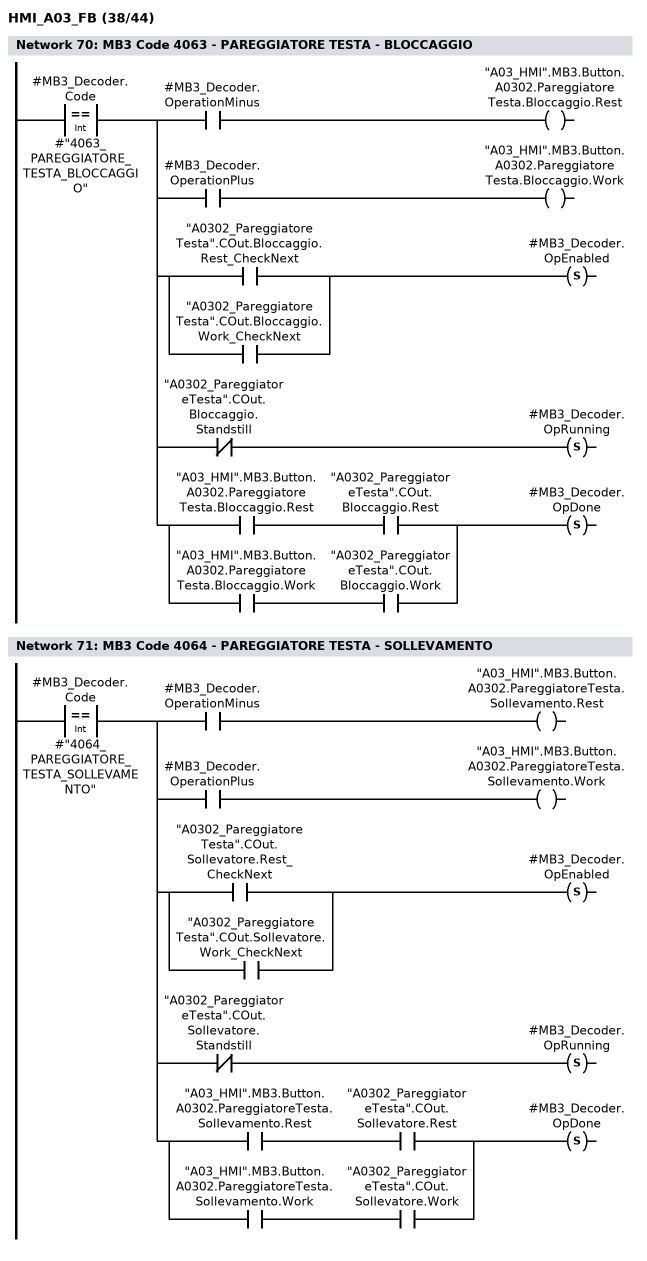
   RUNG wire#powerrail
      { S7_Templates := "SrcType := Int" } EQ_Contact(in1 := #MB3_Decoder.Code, in2 := #"4063_PAREGGIATORE_TESTA_BLOCCAGGIO")
      wire#w1
      Contact( #MB3_Decoder.OperationMinus )
      Coil( "A03_HMI".MB3.Button.A0302.PareggiatoreTesta.Bloccaggio.Rest )
   END_RUNG
   RUNG wire#w1
      Contact( #MB3_Decoder.OperationPlus )
      Coil( "A03_HMI".MB3.Button.A0302.PareggiatoreTesta.Bloccaggio.Work )
   END_RUNG
   RUNG wire#w1
      Contact( "A0302_PareggiatoreTesta".COut.Bloccaggio.Rest_CheckNext )
      wire#w2
      S_Coil( #MB3_Decoder.OpEnabled )
   END_RUNG
   RUNG wire#w1
      Contact( "A0302_PareggiatoreTesta".COut.Bloccaggio.Work_CheckNext )
   END_RUNG wire#w2
   RUNG wire#w1
      I_Contact( "A0302_PareggiatoreTesta".COut.Bloccaggio.Standstill )
      S_Coil( #MB3_Decoder.OpRunning )
   END_RUNG
   RUNG wire#w1
      Contact( "A03_HMI".MB3.Button.A0302.PareggiatoreTesta.Bloccaggio.Rest )
      Contact( "A0302_PareggiatoreTesta".COut.Bloccaggio.Rest )
      wire#w3
      S_Coil( #MB3_Decoder.OpDone )
   END_RUNG
   RUNG wire#w1
      Contact( "A03_HMI".MB3.Button.A0302.PareggiatoreTesta.Bloccaggio.Work )
      Contact( "A0302_PareggiatoreTesta".COut.Bloccaggio.Work )
   END_RUNG wire#w3
   // the same network as SCL:
   #_w1 := #MB3_Decoder.Code = #"4063_PAREGGIATORE_TESTA_BLOCCAGGIO";
   "A03_HMI".MB3.Button.A0302.PareggiatoreTesta.Bloccaggio.Rest := #_w1 AND #MB3_Decoder.OperationMinus;
   "A03_HMI".MB3.Button.A0302.PareggiatoreTesta.Bloccaggio.Work := #_w1 AND #MB3_Decoder.OperationPlus;
   IF #_w1 AND ("A0302_PareggiatoreTesta".COut.Bloccaggio.Rest_CheckNext OR "A0302_PareggiatoreTesta".COut.Bloccaggio.Work_CheckNext) THEN
       #MB3_Decoder.OpEnabled := TRUE;
   END_IF;
   IF #_w1 AND NOT "A0302_PareggiatoreTesta".COut.Bloccaggio.Standstill THEN
       #MB3_Decoder.OpRunning := TRUE;
   END_IF;
   IF #_w1 AND (("A03_HMI".MB3.Button.A0302.PareggiatoreTesta.Bloccaggio.Rest AND "A0302_PareggiatoreTesta".COut.Bloccaggio.Rest) OR ("A03_HMI".MB3.Button.A0302.PareggiatoreTesta.Bloccaggio.Work AND "A0302_PareggiatoreTesta".COut.Bloccaggio.Work)) THEN
       #MB3_Decoder.OpDone := TRUE;
   END_IF;
END_REGION

REGION Network 71: MB3 Code 4064 - PAREGGIATORE TESTA - SOLLEVAMENTO
   RUNG wire#powerrail
      { S7_Templates := "SrcType := Int" } EQ_Contact(in1 := #MB3_Decoder.Code, in2 := #"4064_PAREGGIATORE_TESTA_SOLLEVAMENTO")
      wire#w1
      Contact( #MB3_Decoder.OperationMinus )
      Coil( "A03_HMI".MB3.Button.A0302.PareggiatoreTesta.Sollevamento.Rest )
   END_RUNG
   RUNG wire#w1
      Contact( #MB3_Decoder.OperationPlus )
      Coil( "A03_HMI".MB3.Button.A0302.PareggiatoreTesta.Sollevamento.Work )
   END_RUNG
   RUNG wire#w1
      Contact( "A0302_PareggiatoreTesta".COut.Sollevatore.Rest_CheckNext )
      wire#w2
      S_Coil( #MB3_Decoder.OpEnabled )
   END_RUNG
   RUNG wire#w1
      Contact( "A0302_PareggiatoreTesta".COut.Sollevatore.Work_CheckNext )
   END_RUNG wire#w2
   RUNG wire#w1
      I_Contact( "A0302_PareggiatoreTesta".COut.Sollevatore.Standstill )
      S_Coil( #MB3_Decoder.OpRunning )
   END_RUNG
   RUNG wire#w1
      Contact( "A03_HMI".MB3.Button.A0302.PareggiatoreTesta.Sollevamento.Rest )
      Contact( "A0302_PareggiatoreTesta".COut.Sollevatore.Rest )
      wire#w3
      S_Coil( #MB3_Decoder.OpDone )
   END_RUNG
   RUNG wire#w1
      Contact( "A03_HMI".MB3.Button.A0302.PareggiatoreTesta.Sollevamento.Work )
      Contact( "A0302_PareggiatoreTesta".COut.Sollevatore.Work )
   END_RUNG wire#w3
   // the same network as SCL:
   #_w1 := #MB3_Decoder.Code = #"4064_PAREGGIATORE_TESTA_SOLLEVAMENTO";
   "A03_HMI".MB3.Button.A0302.PareggiatoreTesta.Sollevamento.Rest := #_w1 AND #MB3_Decoder.OperationMinus;
   "A03_HMI".MB3.Button.A0302.PareggiatoreTesta.Sollevamento.Work := #_w1 AND #MB3_Decoder.OperationPlus;
   IF #_w1 AND ("A0302_PareggiatoreTesta".COut.Sollevatore.Rest_CheckNext OR "A0302_PareggiatoreTesta".COut.Sollevatore.Work_CheckNext) THEN
       #MB3_Decoder.OpEnabled := TRUE;
   END_IF;
   IF #_w1 AND NOT "A0302_PareggiatoreTesta".COut.Sollevatore.Standstill THEN
       #MB3_Decoder.OpRunning := TRUE;
   END_IF;
   IF #_w1 AND (("A03_HMI".MB3.Button.A0302.PareggiatoreTesta.Sollevamento.Rest AND "A0302_PareggiatoreTesta".COut.Sollevatore.Rest) OR ("A03_HMI".MB3.Button.A0302.PareggiatoreTesta.Sollevamento.Work AND "A0302_PareggiatoreTesta".COut.Sollevatore.Work)) THEN
       #MB3_Decoder.OpDone := TRUE;
   END_IF;
END_REGION

REGION Network 72: MB3 Code 4064 - PAREGGIATORE TESTA - CENTRAGGIO
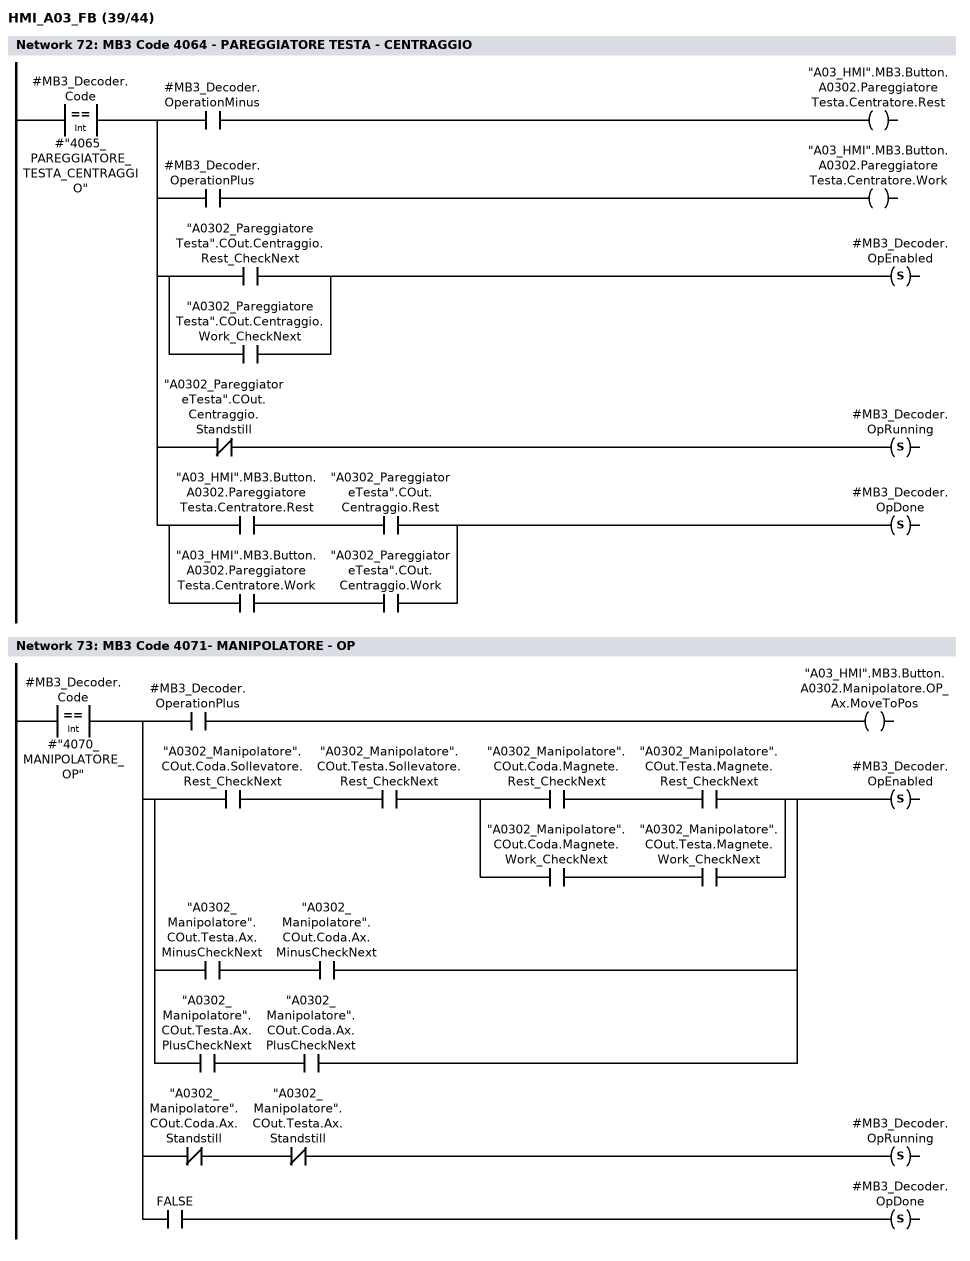
   RUNG wire#powerrail
      { S7_Templates := "SrcType := Int" } EQ_Contact(in1 := #MB3_Decoder.Code, in2 := #"4065_PAREGGIATORE_TESTA_CENTRAGGIO")
      wire#w1
      Contact( #MB3_Decoder.OperationMinus )
      Coil( "A03_HMI".MB3.Button.A0302.PareggiatoreTesta.Centratore.Rest )
   END_RUNG
   RUNG wire#w1
      Contact( #MB3_Decoder.OperationPlus )
      Coil( "A03_HMI".MB3.Button.A0302.PareggiatoreTesta.Centratore.Work )
   END_RUNG
   RUNG wire#w1
      Contact( "A0302_PareggiatoreTesta".COut.Centraggio.Rest_CheckNext )
      wire#w2
      S_Coil( #MB3_Decoder.OpEnabled )
   END_RUNG
   RUNG wire#w1
      Contact( "A0302_PareggiatoreTesta".COut.Centraggio.Work_CheckNext )
   END_RUNG wire#w2
   RUNG wire#w1
      I_Contact( "A0302_PareggiatoreTesta".COut.Centraggio.Standstill )
      S_Coil( #MB3_Decoder.OpRunning )
   END_RUNG
   RUNG wire#w1
      Contact( "A03_HMI".MB3.Button.A0302.PareggiatoreTesta.Centratore.Rest )
      Contact( "A0302_PareggiatoreTesta".COut.Centraggio.Rest )
      wire#w3
      S_Coil( #MB3_Decoder.OpDone )
   END_RUNG
   RUNG wire#w1
      Contact( "A03_HMI".MB3.Button.A0302.PareggiatoreTesta.Centratore.Work )
      Contact( "A0302_PareggiatoreTesta".COut.Centraggio.Work )
   END_RUNG wire#w3
   // the same network as SCL:
   #_w1 := #MB3_Decoder.Code = #"4065_PAREGGIATORE_TESTA_CENTRAGGIO";
   "A03_HMI".MB3.Button.A0302.PareggiatoreTesta.Centratore.Rest := #_w1 AND #MB3_Decoder.OperationMinus;
   "A03_HMI".MB3.Button.A0302.PareggiatoreTesta.Centratore.Work := #_w1 AND #MB3_Decoder.OperationPlus;
   IF #_w1 AND ("A0302_PareggiatoreTesta".COut.Centraggio.Rest_CheckNext OR "A0302_PareggiatoreTesta".COut.Centraggio.Work_CheckNext) THEN
       #MB3_Decoder.OpEnabled := TRUE;
   END_IF;
   IF #_w1 AND NOT "A0302_PareggiatoreTesta".COut.Centraggio.Standstill THEN
       #MB3_Decoder.OpRunning := TRUE;
   END_IF;
   IF #_w1 AND (("A03_HMI".MB3.Button.A0302.PareggiatoreTesta.Centratore.Rest AND "A0302_PareggiatoreTesta".COut.Centraggio.Rest) OR ("A03_HMI".MB3.Button.A0302.PareggiatoreTesta.Centratore.Work AND "A0302_PareggiatoreTesta".COut.Centraggio.Work)) THEN
       #MB3_Decoder.OpDone := TRUE;
   END_IF;
END_REGION

REGION Network 73: MB3 Code 4071- MANIPOLATORE - OP
   RUNG wire#powerrail
      { S7_Templates := "SrcType := Int" } EQ_Contact(in1 := #MB3_Decoder.Code, in2 := #"4070_MANIPOLATORE_OP")
      wire#w1
      Contact( #MB3_Decoder.OperationPlus )
      Coil( "A03_HMI".MB3.Button.A0302.Manipolatore.OP_Ax.MoveToPos )
   END_RUNG
   RUNG wire#w1
      Contact( "A0302_Manipolatore".COut.Coda.Sollevatore.Rest_CheckNext )
      Contact( "A0302_Manipolatore".COut.Testa.Sollevatore.Rest_CheckNext )
      wire#w2
      Contact( "A0302_Manipolatore".COut.Coda.Magnete.Rest_CheckNext )
      Contact( "A0302_Manipolatore".COut.Testa.Magnete.Rest_CheckNext )
      wire#w3
      S_Coil( #MB3_Decoder.OpEnabled )
   END_RUNG
   RUNG wire#w2
      Contact( "A0302_Manipolatore".COut.Coda.Magnete.Work_CheckNext )
      Contact( "A0302_Manipolatore".COut.Testa.Magnete.Work_CheckNext )
   END_RUNG wire#w3
   RUNG wire#w1
      Contact( "A0302_Manipolatore".COut.Testa.Ax.MinusCheckNext )
      Contact( "A0302_Manipolatore".COut.Coda.Ax.MinusCheckNext )
   END_RUNG wire#w3
   RUNG wire#w1
      Contact( "A0302_Manipolatore".COut.Testa.Ax.PlusCheckNext )
      Contact( "A0302_Manipolatore".COut.Coda.Ax.PlusCheckNext )
   END_RUNG wire#w3
   RUNG wire#w1
      I_Contact( "A0302_Manipolatore".COut.Coda.Ax.Standstill )
      I_Contact( "A0302_Manipolatore".COut.Testa.Ax.Standstill )
      S_Coil( #MB3_Decoder.OpRunning )
   END_RUNG
   RUNG wire#w1
      Contact( FALSE )
      S_Coil( #MB3_Decoder.OpDone )
   END_RUNG
   // the same network as SCL:
   #_w1 := #MB3_Decoder.Code = #"4070_MANIPOLATORE_OP";
   "A03_HMI".MB3.Button.A0302.Manipolatore.OP_Ax.MoveToPos := #_w1 AND #MB3_Decoder.OperationPlus;
   IF #_w1 AND (("A0302_Manipolatore".COut.Coda.Sollevatore.Rest_CheckNext AND "A0302_Manipolatore".COut.Testa.Sollevatore.Rest_CheckNext AND (("A0302_Manipolatore".COut.Coda.Magnete.Rest_CheckNext AND "A0302_Manipolatore".COut.Testa.Magnete.Rest_CheckNext) OR ("A0302_Manipolatore".COut.Coda.Magnete.Work_CheckNext AND "A0302_Manipolatore".COut.Testa.Magnete.Work_CheckNext))) OR ("A0302_Manipolatore".COut.Testa.Ax.MinusCheckNext AND "A0302_Manipolatore".COut.Coda.Ax.MinusCheckNext) OR ("A0302_Manipolatore".COut.Testa.Ax.PlusCheckNext AND "A0302_Manipolatore".COut.Coda.Ax.PlusCheckNext)) THEN
       #MB3_Decoder.OpEnabled := TRUE;
   END_IF;
   IF #_w1 AND NOT "A0302_Manipolatore".COut.Coda.Ax.Standstill AND NOT "A0302_Manipolatore".COut.Testa.Ax.Standstill THEN
       #MB3_Decoder.OpRunning := TRUE;
   END_IF;
   IF #_w1 AND FALSE THEN #MB3_Decoder.OpDone := TRUE; END_IF;
END_REGION

REGION Network 74: MB3 Code 4071- MANIPOLATORE -AX
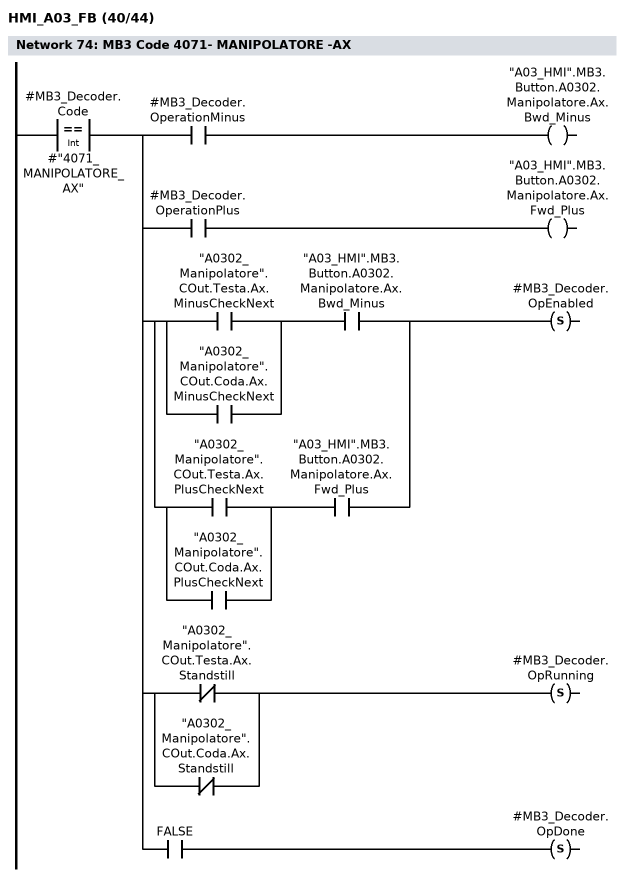
   RUNG wire#powerrail
      { S7_Templates := "SrcType := Int" } EQ_Contact(in1 := #MB3_Decoder.Code, in2 := #"4071_MANIPOLATORE_AX")
      wire#w1
      Contact( #MB3_Decoder.OperationMinus )
      Coil( "A03_HMI".MB3.Button.A0302.Manipolatore.Ax.Bwd_Minus )
   END_RUNG
   RUNG wire#w1
      Contact( #MB3_Decoder.OperationPlus )
      Coil( "A03_HMI".MB3.Button.A0302.Manipolatore.Ax.Fwd_Plus )
   END_RUNG
   RUNG wire#w1
      Contact( "A0302_Manipolatore".COut.Testa.Ax.MinusCheckNext )
      wire#w2
      Contact( "A03_HMI".MB3.Button.A0302.Manipolatore.Ax.Bwd_Minus )
      wire#w3
      S_Coil( #MB3_Decoder.OpEnabled )
   END_RUNG
   RUNG wire#w1
      Contact( "A0302_Manipolatore".COut.Coda.Ax.MinusCheckNext )
   END_RUNG wire#w2
   RUNG wire#w1
      Contact( "A0302_Manipolatore".COut.Testa.Ax.PlusCheckNext )
      wire#w4
      Contact( "A03_HMI".MB3.Button.A0302.Manipolatore.Ax.Fwd_Plus )
   END_RUNG wire#w3
   RUNG wire#w1
      Contact( "A0302_Manipolatore".COut.Coda.Ax.PlusCheckNext )
   END_RUNG wire#w4
   RUNG wire#w1
      I_Contact( "A0302_Manipolatore".COut.Testa.Ax.Standstill )
      wire#w5
      S_Coil( #MB3_Decoder.OpRunning )
   END_RUNG
   RUNG wire#w1
      I_Contact( "A0302_Manipolatore".COut.Coda.Ax.Standstill )
   END_RUNG wire#w5
   RUNG wire#w1
      Contact( FALSE )
      S_Coil( #MB3_Decoder.OpDone )
   END_RUNG
   // the same network as SCL:
   #_w1 := #MB3_Decoder.Code = #"4071_MANIPOLATORE_AX";
   "A03_HMI".MB3.Button.A0302.Manipolatore.Ax.Bwd_Minus := #_w1 AND #MB3_Decoder.OperationMinus;
   "A03_HMI".MB3.Button.A0302.Manipolatore.Ax.Fwd_Plus := #_w1 AND #MB3_Decoder.OperationPlus;
   IF #_w1 AND ((("A0302_Manipolatore".COut.Testa.Ax.MinusCheckNext OR "A0302_Manipolatore".COut.Coda.Ax.MinusCheckNext) AND "A03_HMI".MB3.Button.A0302.Manipolatore.Ax.Bwd_Minus) OR (("A0302_Manipolatore".COut.Testa.Ax.PlusCheckNext OR "A0302_Manipolatore".COut.Coda.Ax.PlusCheckNext) AND "A03_HMI".MB3.Button.A0302.Manipolatore.Ax.Fwd_Plus)) THEN
       #MB3_Decoder.OpEnabled := TRUE;
   END_IF;
   IF #_w1 AND (NOT "A0302_Manipolatore".COut.Testa.Ax.Standstill OR NOT "A0302_Manipolatore".COut.Coda.Ax.Standstill) THEN
       #MB3_Decoder.OpRunning := TRUE;
   END_IF;
   IF #_w1 AND FALSE THEN #MB3_Decoder.OpDone := TRUE; END_IF;
END_REGION

REGION Network 75: MB3 Code 4072- MANIPOLATORE -AX-POS
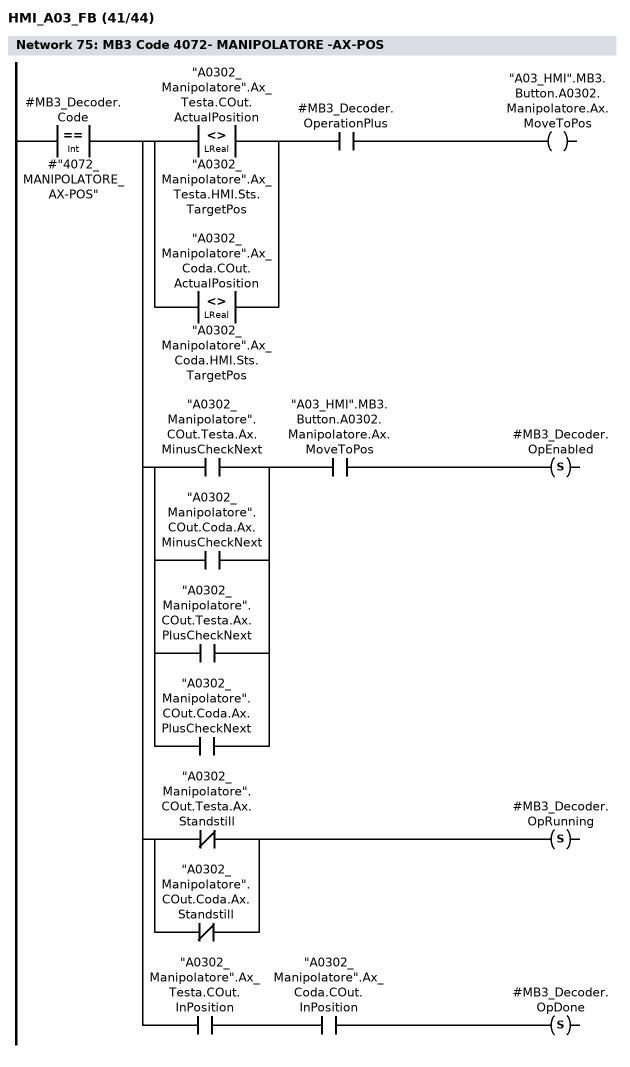
   RUNG wire#powerrail
      { S7_Templates := "SrcType := Int" } EQ_Contact(in1 := #MB3_Decoder.Code, in2 := #"4072_MANIPOLATORE_AX-POS")
      wire#w1
      { S7_Templates := "SrcType := LReal" } NE_Contact(in1 := "A0302_Manipolatore".Ax_Testa.COut.ActualPosition, in2 := "A0302_Manipolatore".Ax_Testa.HMI.Sts.TargetPos)
      wire#w2
      Contact( #MB3_Decoder.OperationPlus )
      Coil( "A03_HMI".MB3.Button.A0302.Manipolatore.Ax.MoveToPos )
   END_RUNG
   RUNG wire#w1
      { S7_Templates := "SrcType := LReal" } NE_Contact(in1 := "A0302_Manipolatore".Ax_Coda.COut.ActualPosition, in2 := "A0302_Manipolatore".Ax_Coda.HMI.Sts.TargetPos)
   END_RUNG wire#w2
   RUNG wire#w1
      Contact( "A0302_Manipolatore".COut.Testa.Ax.MinusCheckNext )
      wire#w3
      Contact( "A03_HMI".MB3.Button.A0302.Manipolatore.Ax.MoveToPos )
      S_Coil( #MB3_Decoder.OpEnabled )
   END_RUNG
   RUNG wire#w1
      Contact( "A0302_Manipolatore".COut.Coda.Ax.MinusCheckNext )
   END_RUNG wire#w3
   RUNG wire#w1
      Contact( "A0302_Manipolatore".COut.Testa.Ax.PlusCheckNext )
   END_RUNG wire#w3
   RUNG wire#w1
      Contact( "A0302_Manipolatore".COut.Coda.Ax.PlusCheckNext )
   END_RUNG wire#w3
   RUNG wire#w1
      I_Contact( "A0302_Manipolatore".COut.Testa.Ax.Standstill )
      wire#w4
      S_Coil( #MB3_Decoder.OpRunning )
   END_RUNG
   RUNG wire#w1
      I_Contact( "A0302_Manipolatore".COut.Coda.Ax.Standstill )
   END_RUNG wire#w4
   RUNG wire#w1
      Contact( "A0302_Manipolatore".Ax_Testa.COut.InPosition )
      Contact( "A0302_Manipolatore".Ax_Coda.COut.InPosition )
      S_Coil( #MB3_Decoder.OpDone )
   END_RUNG
   // the same network as SCL:
   #_w1 := #MB3_Decoder.Code = #"4072_MANIPOLATORE_AX-POS";
   "A03_HMI".MB3.Button.A0302.Manipolatore.Ax.MoveToPos := #_w1 AND (("A0302_Manipolatore".Ax_Testa.COut.ActualPosition <> "A0302_Manipolatore".Ax_Testa.HMI.Sts.TargetPos) OR ("A0302_Manipolatore".Ax_Coda.COut.ActualPosition <> "A0302_Manipolatore".Ax_Coda.HMI.Sts.TargetPos)) AND #MB3_Decoder.OperationPlus;
   IF #_w1 AND ("A0302_Manipolatore".COut.Testa.Ax.MinusCheckNext OR "A0302_Manipolatore".COut.Coda.Ax.MinusCheckNext OR "A0302_Manipolatore".COut.Testa.Ax.PlusCheckNext OR "A0302_Manipolatore".COut.Coda.Ax.PlusCheckNext) AND "A03_HMI".MB3.Button.A0302.Manipolatore.Ax.MoveToPos THEN
       #MB3_Decoder.OpEnabled := TRUE;
   END_IF;
   IF #_w1 AND (NOT "A0302_Manipolatore".COut.Testa.Ax.Standstill OR NOT "A0302_Manipolatore".COut.Coda.Ax.Standstill) THEN
       #MB3_Decoder.OpRunning := TRUE;
   END_IF;
   IF #_w1 AND "A0302_Manipolatore".Ax_Testa.COut.InPosition AND "A0302_Manipolatore".Ax_Coda.COut.InPosition THEN
       #MB3_Decoder.OpDone := TRUE;
   END_IF;
END_REGION

REGION Network 76: MB3 Code 4073 - MANIPOLATORE- MAGNETE
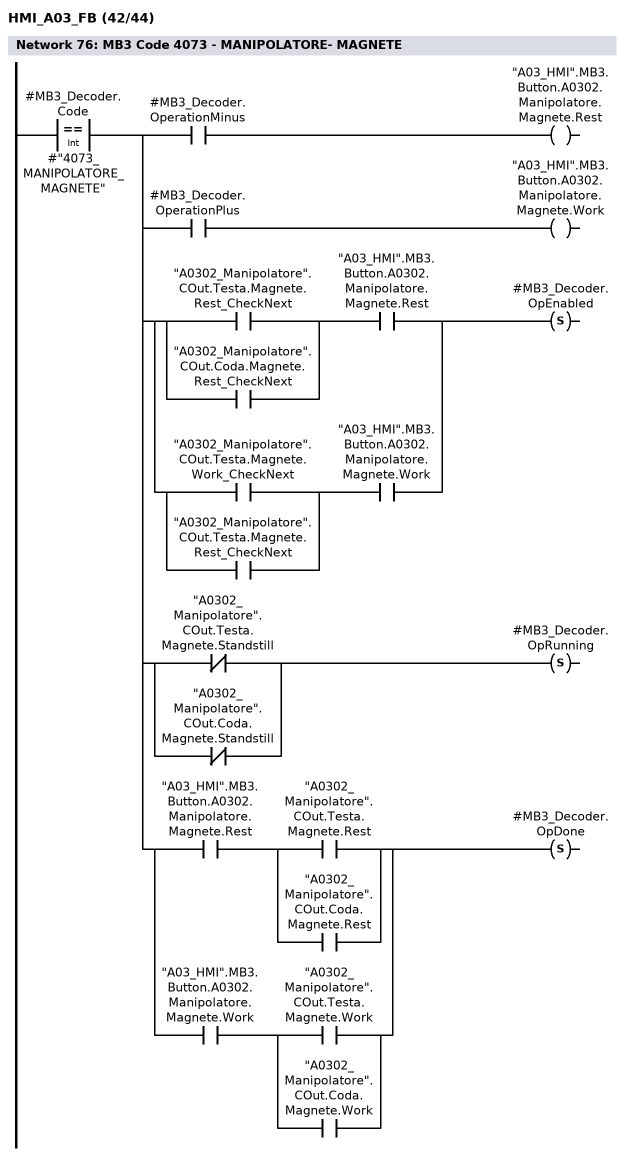
   RUNG wire#powerrail
      { S7_Templates := "SrcType := Int" } EQ_Contact(in1 := #MB3_Decoder.Code, in2 := #"4073_MANIPOLATORE_MAGNETE")
      wire#w1
      Contact( #MB3_Decoder.OperationMinus )
      Coil( "A03_HMI".MB3.Button.A0302.Manipolatore.Magnete.Rest )
   END_RUNG
   RUNG wire#w1
      Contact( #MB3_Decoder.OperationPlus )
      Coil( "A03_HMI".MB3.Button.A0302.Manipolatore.Magnete.Work )
   END_RUNG
   RUNG wire#w1
      Contact( "A0302_Manipolatore".COut.Testa.Magnete.Rest_CheckNext )
      wire#w2
      Contact( "A03_HMI".MB3.Button.A0302.Manipolatore.Magnete.Rest )
      wire#w3
      S_Coil( #MB3_Decoder.OpEnabled )
   END_RUNG
   RUNG wire#w1
      Contact( "A0302_Manipolatore".COut.Coda.Magnete.Rest_CheckNext )
   END_RUNG wire#w2
   RUNG wire#w1
      Contact( "A0302_Manipolatore".COut.Testa.Magnete.Work_CheckNext )
      wire#w4
      Contact( "A03_HMI".MB3.Button.A0302.Manipolatore.Magnete.Work )
   END_RUNG wire#w3
   RUNG wire#w1
      Contact( "A0302_Manipolatore".COut.Testa.Magnete.Rest_CheckNext )
   END_RUNG wire#w4
   RUNG wire#w1
      I_Contact( "A0302_Manipolatore".COut.Testa.Magnete.Standstill )
      wire#w5
      S_Coil( #MB3_Decoder.OpRunning )
   END_RUNG
   RUNG wire#w1
      I_Contact( "A0302_Manipolatore".COut.Coda.Magnete.Standstill )
   END_RUNG wire#w5
   RUNG wire#w1
      Contact( "A03_HMI".MB3.Button.A0302.Manipolatore.Magnete.Rest )
      wire#w6
      Contact( "A0302_Manipolatore".COut.Testa.Magnete.Rest )
      wire#w7
      S_Coil( #MB3_Decoder.OpDone )
   END_RUNG
   RUNG wire#w6
      Contact( "A0302_Manipolatore".COut.Coda.Magnete.Rest )
   END_RUNG wire#w7
   RUNG wire#w1
      Contact( "A03_HMI".MB3.Button.A0302.Manipolatore.Magnete.Work )
      wire#w8
      Contact( "A0302_Manipolatore".COut.Testa.Magnete.Work )
   END_RUNG wire#w7
   RUNG wire#w8
      Contact( "A0302_Manipolatore".COut.Coda.Magnete.Work )
   END_RUNG wire#w7
   // the same network as SCL:
   #_w1 := #MB3_Decoder.Code = #"4073_MANIPOLATORE_MAGNETE";
   "A03_HMI".MB3.Button.A0302.Manipolatore.Magnete.Rest := #_w1 AND #MB3_Decoder.OperationMinus;
   "A03_HMI".MB3.Button.A0302.Manipolatore.Magnete.Work := #_w1 AND #MB3_Decoder.OperationPlus;
   IF #_w1 AND ((("A0302_Manipolatore".COut.Testa.Magnete.Rest_CheckNext OR "A0302_Manipolatore".COut.Coda.Magnete.Rest_CheckNext) AND "A03_HMI".MB3.Button.A0302.Manipolatore.Magnete.Rest) OR (("A0302_Manipolatore".COut.Testa.Magnete.Work_CheckNext OR "A0302_Manipolatore".COut.Testa.Magnete.Rest_CheckNext) AND "A03_HMI".MB3.Button.A0302.Manipolatore.Magnete.Work)) THEN
       #MB3_Decoder.OpEnabled := TRUE;
   END_IF;
   IF #_w1 AND (NOT "A0302_Manipolatore".COut.Testa.Magnete.Standstill OR NOT "A0302_Manipolatore".COut.Coda.Magnete.Standstill) THEN
       #MB3_Decoder.OpRunning := TRUE;
   END_IF;
   IF #_w1 AND (("A03_HMI".MB3.Button.A0302.Manipolatore.Magnete.Rest AND ("A0302_Manipolatore".COut.Testa.Magnete.Rest OR "A0302_Manipolatore".COut.Coda.Magnete.Rest)) OR ("A03_HMI".MB3.Button.A0302.Manipolatore.Magnete.Work AND ("A0302_Manipolatore".COut.Testa.Magnete.Work OR "A0302_Manipolatore".COut.Coda.Magnete.Work))) THEN
       #MB3_Decoder.OpDone := TRUE;
   END_IF;
END_REGION

REGION Network 77: MB3 Code 4074 - MANIPOLATORE- SOLLEVATORE
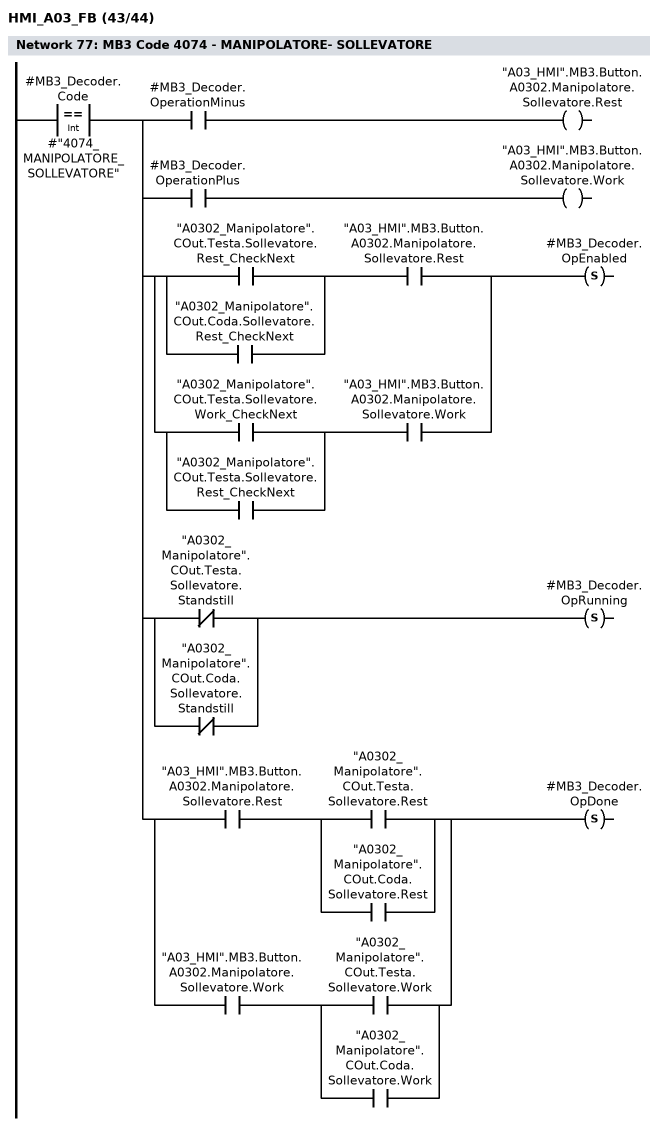
   RUNG wire#powerrail
      { S7_Templates := "SrcType := Int" } EQ_Contact(in1 := #MB3_Decoder.Code, in2 := #"4074_MANIPOLATORE_SOLLEVATORE")
      wire#w1
      Contact( #MB3_Decoder.OperationMinus )
      Coil( "A03_HMI".MB3.Button.A0302.Manipolatore.Sollevatore.Rest )
   END_RUNG
   RUNG wire#w1
      Contact( #MB3_Decoder.OperationPlus )
      Coil( "A03_HMI".MB3.Button.A0302.Manipolatore.Sollevatore.Work )
   END_RUNG
   RUNG wire#w1
      Contact( "A0302_Manipolatore".COut.Testa.Sollevatore.Rest_CheckNext )
      wire#w2
      Contact( "A03_HMI".MB3.Button.A0302.Manipolatore.Sollevatore.Rest )
      wire#w3
      S_Coil( #MB3_Decoder.OpEnabled )
   END_RUNG
   RUNG wire#w1
      Contact( "A0302_Manipolatore".COut.Coda.Sollevatore.Rest_CheckNext )
   END_RUNG wire#w2
   RUNG wire#w1
      Contact( "A0302_Manipolatore".COut.Testa.Sollevatore.Work_CheckNext )
      wire#w4
      Contact( "A03_HMI".MB3.Button.A0302.Manipolatore.Sollevatore.Work )
   END_RUNG wire#w3
   RUNG wire#w1
      Contact( "A0302_Manipolatore".COut.Testa.Sollevatore.Rest_CheckNext )
   END_RUNG wire#w4
   RUNG wire#w1
      I_Contact( "A0302_Manipolatore".COut.Testa.Sollevatore.Standstill )
      wire#w5
      S_Coil( #MB3_Decoder.OpRunning )
   END_RUNG
   RUNG wire#w1
      I_Contact( "A0302_Manipolatore".COut.Coda.Sollevatore.Standstill )
   END_RUNG wire#w5
   RUNG wire#w1
      Contact( "A03_HMI".MB3.Button.A0302.Manipolatore.Sollevatore.Rest )
      wire#w6
      Contact( "A0302_Manipolatore".COut.Testa.Sollevatore.Rest )
      wire#w7
      S_Coil( #MB3_Decoder.OpDone )
   END_RUNG
   RUNG wire#w6
      Contact( "A0302_Manipolatore".COut.Coda.Sollevatore.Rest )
   END_RUNG wire#w7
   RUNG wire#w1
      Contact( "A03_HMI".MB3.Button.A0302.Manipolatore.Sollevatore.Work )
      wire#w8
      Contact( "A0302_Manipolatore".COut.Testa.Sollevatore.Work )
   END_RUNG wire#w7
   RUNG wire#w8
      Contact( "A0302_Manipolatore".COut.Coda.Sollevatore.Work )
   END_RUNG wire#w7
   // the same network as SCL:
   #_w1 := #MB3_Decoder.Code = #"4074_MANIPOLATORE_SOLLEVATORE";
   "A03_HMI".MB3.Button.A0302.Manipolatore.Sollevatore.Rest := #_w1 AND #MB3_Decoder.OperationMinus;
   "A03_HMI".MB3.Button.A0302.Manipolatore.Sollevatore.Work := #_w1 AND #MB3_Decoder.OperationPlus;
   IF #_w1 AND ((("A0302_Manipolatore".COut.Testa.Sollevatore.Rest_CheckNext OR "A0302_Manipolatore".COut.Coda.Sollevatore.Rest_CheckNext) AND "A03_HMI".MB3.Button.A0302.Manipolatore.Sollevatore.Rest) OR (("A0302_Manipolatore".COut.Testa.Sollevatore.Work_CheckNext OR "A0302_Manipolatore".COut.Testa.Sollevatore.Rest_CheckNext) AND "A03_HMI".MB3.Button.A0302.Manipolatore.Sollevatore.Work)) THEN
       #MB3_Decoder.OpEnabled := TRUE;
   END_IF;
   IF #_w1 AND (NOT "A0302_Manipolatore".COut.Testa.Sollevatore.Standstill OR NOT "A0302_Manipolatore".COut.Coda.Sollevatore.Standstill) THEN
       #MB3_Decoder.OpRunning := TRUE;
   END_IF;
   IF #_w1 AND (("A03_HMI".MB3.Button.A0302.Manipolatore.Sollevatore.Rest AND ("A0302_Manipolatore".COut.Testa.Sollevatore.Rest OR "A0302_Manipolatore".COut.Coda.Sollevatore.Rest)) OR ("A03_HMI".MB3.Button.A0302.Manipolatore.Sollevatore.Work AND ("A0302_Manipolatore".COut.Testa.Sollevatore.Work OR "A0302_Manipolatore".COut.Coda.Sollevatore.Work))) THEN
       #MB3_Decoder.OpDone := TRUE;
   END_IF;
END_REGION

REGION Network 79: >
END_REGION

REGION Network 80: >
END_REGION

REGION Network 81: >
END_REGION

REGION Network 82: MB3 Decoder
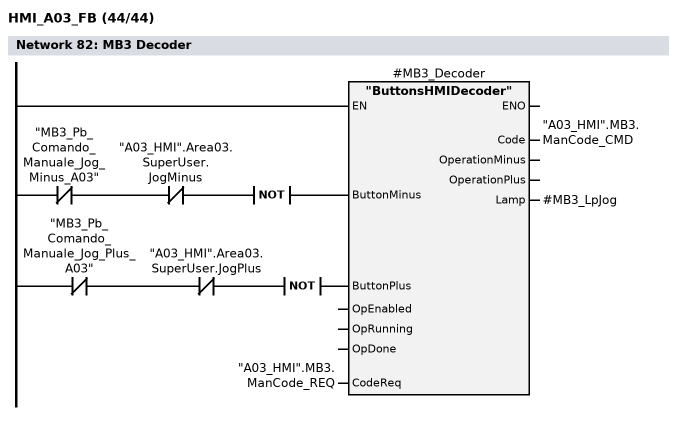
   RUNG wire#powerrail
      #MB3_Decoder(ButtonMinus := wire#w1, ButtonPlus := wire#w2, OpEnabled :=, OpRunning :=, OpDone :=, CodeReq := "A03_HMI".MB3.ManCode_REQ, Code => "A03_HMI".MB3.ManCode_CMD, OperationMinus =>, OperationPlus =>, Lamp => #MB3_LpJog)
   END_RUNG
   RUNG wire#powerrail
      I_Contact( "MB3_Pb_Comando_Manuale_Jog_Minus_A03" )
      I_Contact( "A03_HMI".Area03.SuperUser.JogMinus )
      Not()
   END_RUNG wire#w1
   RUNG wire#powerrail
      I_Contact( "MB3_Pb_Comando_Manuale_Jog_Plus_A03" )
      I_Contact( "A03_HMI".Area03.SuperUser.JogPlus )
      Not()
   END_RUNG wire#w2
   // the same network as SCL:
   #MB3_Decoder(ButtonMinus := NOT (NOT "MB3_Pb_Comando_Manuale_Jog_Minus_A03" AND NOT "A03_HMI".Area03.SuperUser.JogMinus),   // "ButtonsHMIDecoder"
                ButtonPlus := NOT (NOT "MB3_Pb_Comando_Manuale_Jog_Plus_A03" AND NOT "A03_HMI".Area03.SuperUser.JogPlus),
                CodeReq := "A03_HMI".MB3.ManCode_REQ,
                Code => "A03_HMI".MB3.ManCode_CMD,
                Lamp => #MB3_LpJog);
END_REGION
END_FUNCTION_BLOCK
